LIN {X 0,Y 114.864,Z 300.989,A -85,B 0,C 180,E1 -25798.93,E2 -25798.93} C_VEL
LIN {X 0,Y 114.941,Z 300.979,A -85,B 0,C 180,E1 -25806.506,E2 -25806.506} C_VEL
LIN {X 0,Y 115.012,Z 300.965,A -85,B 0,C 180,E1 -25812.209,E2 -25812.209} C_VEL
LIN {X 0,Y 115.278,Z 300.938,A -85,B 0,C 180,E1 -25817.262,E2 -25817.262} C_VEL
LIN {X 0,Y 115.38,Z 300.924,A -85,B 0,C 180,E1 -25823.002,E2 -25823.002} C_VEL
LIN {X 0,Y 115.988,Z 300.845,A -85,B 0,C 180,E1 -25829.999,E2 -25829.999} C_VEL
LIN {X 0,Y 115.381,Z 300.918,A -85,B 0,C 180,E1 -25836.996,E2 -25836.996} C_VEL
LIN {X 0,Y 115.299,Z 300.934,A -85,B 0,C 180,E1 -25842.784,E2 -25842.784} C_VEL
LIN {X 0,Y 115.207,Z 300.943,A -85,B 0,C 180,E1 -25844.122,E2 -25844.122} C_VEL
LIN {X 0,Y 118.06,Z 309.026,A -85,B 0,C 180,E1 -25845.314,E2 -25845.314} C_VEL
LIN {X 0,Y 124.577,Z 328.009,A -85,B 0,C 180,E1 -25847.836,E2 -25847.836} C_VEL
LIN {X 0,Y 122.385,Z 365.038,A -85,B 0,C 180,E1 -25850.533,E2 -25850.533} C_VEL
LIN {X 0,Y 121.452,Z 375.386,A -85,B 0,C 180,E1 -25851.751,E2 -25851.751} C_VEL
LIN {X 0,Y 120.031,Z 387.44,A -85,B 0,C 180,E1 -25853.894,E2 -25853.894} C_VEL
LIN {X 0,Y 118.866,Z 395.437,A -85,B 0,C 180,E1 -25855.788,E2 -25855.788} C_VEL
LIN {X 0,Y 117.488,Z 403.441,A -85,B 0,C 180,E1 -25858.151,E2 -25858.151} C_VEL
LIN {X 0,Y 116.013,Z 411.202,A -85,B 0,C 180,E1 -25860.991,E2 -25860.991} C_VEL
LIN {X 0,Y 114.685,Z 418.966,A -85,B 0,C 180,E1 -25864.529,E2 -25864.529} C_VEL
LIN {X 0,Y 113.39,Z 426.948,A -85,B 0,C 180,E1 -25869.104,E2 -25869.104} C_VEL
LIN {X 0,Y 112.584,Z 432.701,A -85,B 0,C 180,E1 -25873.365,E2 -25873.365} C_VEL
LIN {X 0,Y 112.223,Z 438.256,A -85,B 0,C 180,E1 -25878.718,E2 -25878.718} C_VEL
LIN {X 0,Y 112.358,Z 440.502,A -85,B 0,C 180,E1 -25881.285,E2 -25881.285} C_VEL
LIN {X 0,Y 113.089,Z 443.74,A -85,B 0,C 180,E1 -25885.996,E2 -25885.996} C_VEL
LIN {X 0,Y 114.462,Z 446.022,A -85,B 0,C 180,E1 -25890.584,E2 -25890.584} C_VEL
LIN {X 0,Y 116.506,Z 447.444,A -85,B 0,C 180,E1 -25895.026,E2 -25895.026} C_VEL
LIN {X 0,Y 119.684,Z 448.034,A -85,B 0,C 180,E1 -25899.97,E2 -25899.97} C_VEL
LIN {X 0,Y 123.835,Z 447.495,A -85,B 0,C 180,E1 -25904.745,E2 -25904.745} C_VEL
LIN {X 0,Y 126.367,Z 446.823,A -85,B 0,C 180,E1 -25907.149,E2 -25907.149} C_VEL
LIN {X 0,Y 130.687,Z 445.002,A -85,B 0,C 180,E1 -25910.719,E2 -25910.719} C_VEL
LIN {X 0,Y 135.629,Z 442.26,A -85,B 0,C 180,E1 -25914.054,E2 -25914.054} C_VEL
LIN {X 0,Y 142.473,Z 437.356,A -85,B 0,C 180,E1 -25917.882,E2 -25917.882} C_VEL
LIN {X 0,Y 147.586,Z 432.947,A -85,B 0,C 180,E1 -25920.364,E2 -25920.364} C_VEL
LIN {X 0,Y 152.954,Z 427.55,A -85,B 0,C 180,E1 -25922.636,E2 -25922.636} C_VEL
LIN {X 0,Y 158.242,Z 421.307,A -85,B 0,C 180,E1 -25924.653,E2 -25924.653} C_VEL
LIN {X 0,Y 163.394,Z 414.148,A -85,B 0,C 180,E1 -25926.442,E2 -25926.442} C_VEL
LIN {X 0,Y 168.811,Z 405.171,A -85,B 0,C 180,E1 -25928.163,E2 -25928.163} C_VEL
LIN {X 0,Y 173.777,Z 394.79,A -85,B 0,C 180,E1 -25929.604,E2 -25929.604} C_VEL
LIN {X 0,Y 177.051,Z 385.976,A -85,B 0,C 180,E1 -25930.574,E2 -25930.574} C_VEL
LIN {X 0,Y 179.653,Z 377.072,A -85,B 0,C 180,E1 -25931.282,E2 -25931.282} C_VEL
LIN {X 0,Y 180.084,Z 375.072,A -85,B 0,C 180,E1 -25931.489,E2 -25931.489} C_VEL
LIN {X 0,Y 178.388,Z 370.508,A -85,B 0,C 180,E1 -25935.201,E2 -25935.201} C_VEL
LIN {X 0,Y 177.063,Z 367.237,A -85,B 0,C 180,E1 -25939.365,E2 -25939.365} C_VEL
LIN {X 0,Y 176.416,Z 366.762,A -85,B 0,C 180,E1 -25943.618,E2 -25943.618} C_VEL
LIN {X 0,Y 176.662,Z 367.081,A -85,B 0,C 180,E1 -25946.725,E2 -25946.725} C_VEL
LIN {X 0,Y 177.162,Z 369.122,A -85,B 0,C 180,E1 -25949.713,E2 -25949.713} C_VEL
LIN {X 0,Y 178.163,Z 373.507,A -85,B 0,C 180,E1 -25953.286,E2 -25953.286} C_VEL
LIN {X 0,Y 179.099,Z 377.548,A -85,B 0,C 180,E1 -25955.579,E2 -25955.579} C_VEL
LIN {X 0,Y 179.509,Z 380.366,A -85,B 0,C 180,E1 -25956.937,E2 -25956.937} C_VEL
LIN {X 0,Y 176.688,Z 390.157,A -85,B 0,C 180,E1 -25957.542,E2 -25957.542} C_VEL
LIN {X 0,Y 173.38,Z 398.961,A -85,B 0,C 180,E1 -25958.264,E2 -25958.264} C_VEL
LIN {X 0,Y 169.107,Z 408.204,A -85,B 0,C 180,E1 -25959.284,E2 -25959.284} C_VEL
LIN {X 0,Y 163.498,Z 418.104,A -85,B 0,C 180,E1 -25960.748,E2 -25960.748} C_VEL
LIN {X 0,Y 157.345,Z 426.798,A -85,B 0,C 180,E1 -25962.526,E2 -25962.526} C_VEL
LIN {X 0,Y 152.186,Z 433.149,A -85,B 0,C 180,E1 -25964.294,E2 -25964.294} C_VEL
LIN {X 0,Y 147.242,Z 438.497,A -85,B 0,C 180,E1 -25966.205,E2 -25966.205} C_VEL
LIN {X 0,Y 142.546,Z 443.022,A -85,B 0,C 180,E1 -25968.274,E2 -25968.274} C_VEL
LIN {X 0,Y 135.864,Z 448.445,A -85,B 0,C 180,E1 -25971.632,E2 -25971.632} C_VEL
LIN {X 0,Y 129.891,Z 452.562,A -85,B 0,C 180,E1 -25975.382,E2 -25975.382} C_VEL
LIN {X 0,Y 124.641,Z 455.495,A -85,B 0,C 180,E1 -25979.506,E2 -25979.506} C_VEL
LIN {X 0,Y 121.618,Z 456.789,A -85,B 0,C 180,E1 -25982.466,E2 -25982.466} C_VEL
LIN {X 0,Y 118.968,Z 457.67,A -85,B 0,C 180,E1 -25985.575,E2 -25985.575} C_VEL
LIN {X 0,Y 116.788,Z 458.13,A -85,B 0,C 180,E1 -25988.836,E2 -25988.836} C_VEL
LIN {X 0,Y 115.116,Z 458.028,A -85,B 0,C 180,E1 -25992.228,E2 -25992.228} C_VEL
LIN {X 0,Y 113.962,Z 457.507,A -85,B 0,C 180,E1 -25995.72,E2 -25995.72} C_VEL
LIN {X 0,Y 113.173,Z 456.575,A -85,B 0,C 180,E1 -25999.264,E2 -25999.264} C_VEL
LIN {X 0,Y 112.949,Z 454.232,A -85,B 0,C 180,E1 -26004.627,E2 -26004.627} C_VEL
LIN {X 0,Y 113.104,Z 452.031,A -85,B 0,C 180,E1 -26008.221,E2 -26008.221} C_VEL
LIN {X 0,Y 113.156,Z 449.13,A -85,B 0,C 180,E1 -26011.78,E2 -26011.78} C_VEL
LIN {X 0,Y 113.228,Z 443.223,A -85,B 0,C 180,E1 -26017.132,E2 -26017.132} C_VEL
LIN {X 0,Y 113.61,Z 438.268,A -85,B 0,C 180,E1 -26020.696,E2 -26020.696} C_VEL
LIN {X 0,Y 114.308,Z 432.256,A -85,B 0,C 180,E1 -26024.238,E2 -26024.238} C_VEL
LIN {X 0,Y 115.483,Z 424.969,A -85,B 0,C 180,E1 -26027.716,E2 -26027.716} C_VEL
LIN {X 0,Y 116.861,Z 417.213,A -85,B 0,C 180,E1 -26030.691,E2 -26030.691} C_VEL
LIN {X 0,Y 118.458,Z 407.592,A -85,B 0,C 180,E1 -26033.608,E2 -26033.608} C_VEL
LIN {X 0,Y 120.245,Z 396.823,A -85,B 0,C 180,E1 -26035.999,E2 -26035.999} C_VEL
LIN {X 0,Y 121.486,Z 386.329,A -85,B 0,C 180,E1 -26037.67,E2 -26037.67} C_VEL
LIN {X 0,Y 122.307,Z 377.143,A -85,B 0,C 180,E1 -26038.69,E2 -26038.69} C_VEL
LIN {X 0,Y 123.167,Z 358.274,A -85,B 0,C 180,E1 -26040.134,E2 -26040.134} C_VEL
LIN {X 0,Y 121.253,Z 329.779,A -85,B 0,C 180,E1 -26042.624,E2 -26042.624} C_VEL
LIN {X 0,Y 120.313,Z 326.084,A -85,B 0,C 180,E1 -26043.058,E2 -26043.058} C_VEL
LIN {X 0,Y 116.845,Z 320.753,A -85,B 0,C 180,E1 -26044.039,E2 -26044.039} C_VEL
LIN {X 0,Y 112.972,Z 315.538,A -85,B 0,C 180,E1 -26045.144,E2 -26045.144} C_VEL
LIN {X 0,Y 111.425,Z 311.965,A -85,B 0,C 180,E1 -26045.734,E2 -26045.734} C_VEL
LIN {X 0,Y 109.288,Z 305.743,A -85,B 0,C 180,E1 -26046.684,E2 -26046.684} C_VEL
LIN {X 0,Y 107.873,Z 301.859,A -85,B 0,C 180,E1 -26047.374,E2 -26047.374} C_VEL
LIN {X 0,Y 107.683,Z 301.879,A -85,B 0,C 180,E1 -26054.113,E2 -26054.113} C_VEL
LIN {X 0,Y 107.687,Z 301.877,A -85,B 0,C 180,E1 -26061.551,E2 -26061.551} C_VEL
LIN {X 0,Y 107.795,Z 301.866,A -85,B 0,C 180,E1 -26068.558,E2 -26068.558} C_VEL
LIN {X 0,Y 107.914,Z 301.852,A -85,B 0,C 180,E1 -26076.995,E2 -26076.995} C_VEL
LIN {X 0,Y 108.031,Z 301.839,A -85,B 0,C 180,E1 -26084.914,E2 -26084.914} C_VEL
LIN {X 0,Y 108.256,Z 301.809,A -85,B 0,C 180,E1 -26088.766,E2 -26088.766} C_VEL
LIN {X 0,Y 108.445,Z 301.784,A -85,B 0,C 180,E1 -26096.281,E2 -26096.281} C_VEL
LIN {X 0,Y 108.942,Z 301.727,A -85,B 0,C 180,E1 -26099.997,E2 -26099.997} C_VEL
LIN {X 0,Y 108.327,Z 301.804,A -85,B 0,C 180,E1 -26107.452,E2 -26107.452} C_VEL
LIN {X 0,Y 108.198,Z 301.813,A -85,B 0,C 180,E1 -26113.012,E2 -26113.012} C_VEL
LIN {X 0,Y 107.909,Z 301.854,A -85,B 0,C 180,E1 -26119.001,E2 -26119.001} C_VEL
LIN {X 0,Y 107.858,Z 301.862,A -85,B 0,C 180,E1 -26124.184,E2 -26124.184} C_VEL
LIN {X 0,Y 107.792,Z 301.87,A -85,B 0,C 180,E1 -26132.049,E2 -26132.049} C_VEL
LIN {X 0,Y 107.73,Z 301.872,A -85,B 0,C 180,E1 -26138.478,E2 -26138.478} C_VEL
LIN {X 0,Y 107.763,Z 301.867,A -85,B 0,C 180,E1 -26145.834,E2 -26145.834} C_VEL
LIN {X 0,Y 107.751,Z 301.876,A -85,B 0,C 180,E1 -26151.502,E2 -26151.502} C_VEL
LIN {X 0,Y 107.806,Z 301.868,A -85,B 0,C 180,E1 -26158.565,E2 -26158.565} C_VEL
LIN {X 0,Y 107.905,Z 301.856,A -85,B 0,C 180,E1 -26166.996,E2 -26166.996} C_VEL
LIN {X 0,Y 108.034,Z 301.839,A -85,B 0,C 180,E1 -26174.917,E2 -26174.917} C_VEL
LIN {X 0,Y 108.281,Z 301.805,A -85,B 0,C 180,E1 -26178.771,E2 -26178.771} C_VEL
LIN {X 0,Y 108.449,Z 301.786,A -85,B 0,C 180,E1 -26186.284,E2 -26186.284} C_VEL
LIN {X 0,Y 108.938,Z 301.723,A -85,B 0,C 180,E1 -26189.999,E2 -26189.999} C_VEL
LIN {X 0,Y 108.321,Z 301.797,A -85,B 0,C 180,E1 -26197.455,E2 -26197.455} C_VEL
LIN {X 0,Y 108.241,Z 301.813,A -85,B 0,C 180,E1 -26202.869,E2 -26202.869} C_VEL
LIN {X 0,Y 117.726,Z 329.232,A -85,B 0,C 180,E1 -26206.93,E2 -26206.93} C_VEL
LIN {X 0,Y 115.492,Z 365.51,A -85,B 0,C 180,E1 -26209.722,E2 -26209.722} C_VEL
LIN {X 0,Y 114.416,Z 376.749,A -85,B 0,C 180,E1 -26211.134,E2 -26211.134} C_VEL
LIN {X 0,Y 112.932,Z 388.546,A -85,B 0,C 180,E1 -26213.43,E2 -26213.43} C_VEL
LIN {X 0,Y 111.623,Z 397.143,A -85,B 0,C 180,E1 -26215.66,E2 -26215.66} C_VEL
LIN {X 0,Y 109.955,Z 405.853,A -85,B 0,C 180,E1 -26218.519,E2 -26218.519} C_VEL
LIN {X 0,Y 108.235,Z 415.195,A -85,B 0,C 180,E1 -26222.428,E2 -26222.428} C_VEL
LIN {X 0,Y 106.799,Z 423.439,A -85,B 0,C 180,E1 -26226.974,E2 -26226.974} C_VEL
LIN {X 0,Y 105.92,Z 429.134,A -85,B 0,C 180,E1 -26230.881,E2 -26230.881} C_VEL
LIN {X 0,Y 105.293,Z 434.326,A -85,B 0,C 180,E1 -26235.26,E2 -26235.26} C_VEL
LIN {X 0,Y 105.173,Z 438.298,A -85,B 0,C 180,E1 -26239.349,E2 -26239.349} C_VEL
LIN {X 0,Y 105.484,Z 441.372,A -85,B 0,C 180,E1 -26243.161,E2 -26243.161} C_VEL
LIN {X 0,Y 106.698,Z 444.823,A -85,B 0,C 180,E1 -26248.899,E2 -26248.899} C_VEL
LIN {X 0,Y 108.938,Z 447.125,A -85,B 0,C 180,E1 -26254.576,E2 -26254.576} C_VEL
LIN {X 0,Y 112.177,Z 448.298,A -85,B 0,C 180,E1 -26260.006,E2 -26260.006} C_VEL
LIN {X 0,Y 116.378,Z 448.344,A -85,B 0,C 180,E1 -26265.059,E2 -26265.059} C_VEL
LIN {X 0,Y 121.731,Z 447.128,A -85,B 0,C 180,E1 -26270.029,E2 -26270.029} C_VEL
LIN {X 0,Y 127.18,Z 444.882,A -85,B 0,C 180,E1 -26274.073,E2 -26274.073} C_VEL
LIN {X 0,Y 133.619,Z 441.3,A -85,B 0,C 180,E1 -26277.875,E2 -26277.875} C_VEL
LIN {X 0,Y 140.594,Z 436.359,A -85,B 0,C 180,E1 -26281.344,E2 -26281.344} C_VEL
LIN {X 0,Y 148.024,Z 429.843,A -85,B 0,C 180,E1 -26284.425,E2 -26284.425} C_VEL
LIN {X 0,Y 153.618,Z 423.846,A -85,B 0,C 180,E1 -26286.477,E2 -26286.477} C_VEL
LIN {X 0,Y 158.966,Z 417.122,A -85,B 0,C 180,E1 -26288.264,E2 -26288.264} C_VEL
LIN {X 0,Y 164.281,Z 409.203,A -85,B 0,C 180,E1 -26289.855,E2 -26289.855} C_VEL
LIN {X 0,Y 168.722,Z 401.241,A -85,B 0,C 180,E1 -26291.109,E2 -26291.109} C_VEL
LIN {X 0,Y 172.503,Z 393.028,A -85,B 0,C 180,E1 -26292.106,E2 -26292.106} C_VEL
LIN {X 0,Y 175.803,Z 383.937,A -85,B 0,C 180,E1 -26293.013,E2 -26293.013} C_VEL
LIN {X 0,Y 177.064,Z 379.788,A -85,B 0,C 180,E1 -26293.348,E2 -26293.348} C_VEL
LIN {X 0,Y 176.232,Z 376.932,A -85,B 0,C 180,E1 -26295.994,E2 -26295.994} C_VEL
LIN {X 0,Y 175.527,Z 374.154,A -85,B 0,C 180,E1 -26299.542,E2 -26299.542} C_VEL
LIN {X 0,Y 174.953,Z 373.704,A -85,B 0,C 180,E1 -26303.687,E2 -26303.687} C_VEL
LIN {X 0,Y 175.186,Z 374.126,A -85,B 0,C 180,E1 -26306.708,E2 -26306.708} C_VEL
LIN {X 0,Y 175.475,Z 375.771,A -85,B 0,C 180,E1 -26309.084,E2 -26309.084} C_VEL
LIN {X 0,Y 176.027,Z 379.665,A -85,B 0,C 180,E1 -26312.378,E2 -26312.378} C_VEL
LIN {X 0,Y 176.544,Z 383.979,A -85,B 0,C 180,E1 -26314.894,E2 -26314.894} C_VEL
LIN {X 0,Y 172.323,Z 396.26,A -85,B 0,C 180,E1 -26315.78,E2 -26315.78} C_VEL
LIN {X 0,Y 168.078,Z 405.486,A -85,B 0,C 180,E1 -26316.663,E2 -26316.663} C_VEL
LIN {X 0,Y 163.359,Z 413.939,A -85,B 0,C 180,E1 -26317.768,E2 -26317.768} C_VEL
LIN {X 0,Y 158.303,Z 421.5,A -85,B 0,C 180,E1 -26319.023,E2 -26319.023} C_VEL
LIN {X 0,Y 151.37,Z 430.324,A -85,B 0,C 180,E1 -26321.023,E2 -26321.023} C_VEL
LIN {X 0,Y 144.794,Z 437.322,A -85,B 0,C 180,E1 -26323.278,E2 -26323.278} C_VEL
LIN {X 0,Y 139.815,Z 441.962,A -85,B 0,C 180,E1 -26325.275,E2 -26325.275} C_VEL
LIN {X 0,Y 132.692,Z 447.497,A -85,B 0,C 180,E1 -26328.545,E2 -26328.545} C_VEL
LIN {X 0,Y 126.141,Z 451.703,A -85,B 0,C 180,E1 -26332.204,E2 -26332.204} C_VEL
LIN {X 0,Y 122.164,Z 453.868,A -85,B 0,C 180,E1 -26334.882,E2 -26334.882} C_VEL
LIN {X 0,Y 118.571,Z 455.571,A -85,B 0,C 180,E1 -26337.763,E2 -26337.763} C_VEL
LIN {X 0,Y 115.374,Z 456.695,A -85,B 0,C 180,E1 -26340.837,E2 -26340.837} C_VEL
LIN {X 0,Y 112.549,Z 457.369,A -85,B 0,C 180,E1 -26344.082,E2 -26344.082} C_VEL
LIN {X 0,Y 110.187,Z 457.652,A -85,B 0,C 180,E1 -26347.501,E2 -26347.501} C_VEL
LIN {X 0,Y 108.371,Z 457.513,A -85,B 0,C 180,E1 -26351.081,E2 -26351.081} C_VEL
LIN {X 0,Y 107.114,Z 456.823,A -85,B 0,C 180,E1 -26354.786,E2 -26354.786} C_VEL
LIN {X 0,Y 106.233,Z 455.696,A -85,B 0,C 180,E1 -26358.554,E2 -26358.554} C_VEL
LIN {X 0,Y 105.948,Z 453.139,A -85,B 0,C 180,E1 -26364.305,E2 -26364.305} C_VEL
LIN {X 0,Y 106.133,Z 450.763,A -85,B 0,C 180,E1 -26368.104,E2 -26368.104} C_VEL
LIN {X 0,Y 106.149,Z 447.7,A -85,B 0,C 180,E1 -26371.898,E2 -26371.898} C_VEL
LIN {X 0,Y 106.18,Z 443.174,A -85,B 0,C 180,E1 -26376.266,E2 -26376.266} C_VEL
LIN {X 0,Y 106.545,Z 437.759,A -85,B 0,C 180,E1 -26380.452,E2 -26380.452} C_VEL
LIN {X 0,Y 107.237,Z 431.73,A -85,B 0,C 180,E1 -26384.228,E2 -26384.228} C_VEL
LIN {X 0,Y 108.422,Z 424.419,A -85,B 0,C 180,E1 -26387.933,E2 -26387.933} C_VEL
LIN {X 0,Y 109.848,Z 416.641,A -85,B 0,C 180,E1 -26391.093,E2 -26391.093} C_VEL
LIN {X 0,Y 111.489,Z 406.981,A -85,B 0,C 180,E1 -26394.189,E2 -26394.189} C_VEL
LIN {X 0,Y 113.326,Z 396.093,A -85,B 0,C 180,E1 -26396.719,E2 -26396.719} C_VEL
LIN {X 0,Y 114.559,Z 386.165,A -85,B 0,C 180,E1 -26398.389,E2 -26398.389} C_VEL
LIN {X 0,Y 115.451,Z 376.307,A -85,B 0,C 180,E1 -26399.542,E2 -26399.542} C_VEL
LIN {X 0,Y 116.301,Z 358.488,A -85,B 0,C 180,E1 -26400.978,E2 -26400.978} C_VEL
LIN {X 0,Y 113.92,Z 320.888,A -85,B 0,C 180,E1 -26404.509,E2 -26404.509} C_VEL
LIN {X 0,Y 111.425,Z 311.965,A -85,B 0,C 180,E1 -26405.734,E2 -26405.734} C_VEL
LIN {X 0,Y 110.153,Z 308.851,A -85,B 0,C 180,E1 -26406.532,E2 -26406.532} C_VEL
LIN {X 0,Y 108.481,Z 306.509,A -85,B 0,C 180,E1 -26407.797,E2 -26407.797} C_VEL
LIN {X 0,Y 106.664,Z 304.831,A -85,B 0,C 180,E1 -26409.398,E2 -26409.398} C_VEL
LIN {X 0,Y 104.071,Z 303.42,A -85,B 0,C 180,E1 -26412.26,E2 -26412.26} C_VEL
LIN {X 0,Y 101.917,Z 302.856,A -85,B 0,C 180,E1 -26415.615,E2 -26415.615} C_VEL
LIN {X 0,Y 100.633,Z 302.756,A -85,B 0,C 180,E1 -26420.407,E2 -26420.407} C_VEL
LIN {X 0,Y 100.691,Z 302.754,A -85,B 0,C 180,E1 -26426.884,E2 -26426.884} C_VEL
LIN {X 0,Y 100.789,Z 302.743,A -85,B 0,C 180,E1 -26435.264,E2 -26435.264} C_VEL
LIN {X 0,Y 100.818,Z 302.733,A -85,B 0,C 180,E1 -26439.598,E2 -26439.598} C_VEL
LIN {X 0,Y 101.105,Z 302.696,A -85,B 0,C 180,E1 -26446.696,E2 -26446.696} C_VEL
LIN {X 0,Y 101.243,Z 302.686,A -85,B 0,C 180,E1 -26452.016,E2 -26452.016} C_VEL
LIN {X 0,Y 101.865,Z 302.609,A -85,B 0,C 180,E1 -26459.997,E2 -26459.997} C_VEL
LIN {X 0,Y 101.266,Z 302.684,A -85,B 0,C 180,E1 -26467.975,E2 -26467.975} C_VEL
LIN {X 0,Y 101.123,Z 302.695,A -85,B 0,C 180,E1 -26473.347,E2 -26473.347} C_VEL
LIN {X 0,Y 100.819,Z 302.731,A -85,B 0,C 180,E1 -26480.395,E2 -26480.395} C_VEL
LIN {X 0,Y 100.772,Z 302.745,A -85,B 0,C 180,E1 -26484.955,E2 -26484.955} C_VEL
LIN {X 0,Y 100.699,Z 302.754,A -85,B 0,C 180,E1 -26493.122,E2 -26493.122} C_VEL
LIN {X 0,Y 100.683,Z 302.753,A -85,B 0,C 180,E1 -26499.84,E2 -26499.84} C_VEL
LIN {X 0,Y 100.729,Z 302.743,A -85,B 0,C 180,E1 -26505.756,E2 -26505.756} C_VEL
LIN {X 0,Y 100.691,Z 302.755,A -85,B 0,C 180,E1 -26511.084,E2 -26511.084} C_VEL
LIN {X 0,Y 100.703,Z 302.751,A -85,B 0,C 180,E1 -26516.867,E2 -26516.867} C_VEL
LIN {X 0,Y 100.781,Z 302.741,A -85,B 0,C 180,E1 -26525.265,E2 -26525.265} C_VEL
LIN {X 0,Y 100.812,Z 302.737,A -85,B 0,C 180,E1 -26529.6,E2 -26529.6} C_VEL
LIN {X 0,Y 101.181,Z 302.691,A -85,B 0,C 180,E1 -26537.972,E2 -26537.972} C_VEL
LIN {X 0,Y 101.259,Z 302.681,A -85,B 0,C 180,E1 -26542.02,E2 -26542.02} C_VEL
LIN {X 0,Y 101.862,Z 302.604,A -85,B 0,C 180,E1 -26549.999,E2 -26549.999} C_VEL
LIN {X 0,Y 101.209,Z 302.69,A -85,B 0,C 180,E1 -26559.996,E2 -26559.996} C_VEL
LIN {X 0,Y 101.23,Z 302.695,A -85,B 0,C 180,E1 -26561.512,E2 -26561.512} C_VEL
LIN {X 0,Y 109.715,Z 327.024,A -85,B 0,C 180,E1 -26565.45,E2 -26565.45} C_VEL
LIN {X 0,Y 110.926,Z 330.649,A -85,B 0,C 180,E1 -26565.97,E2 -26565.97} C_VEL
LIN {X 0,Y 108.569,Z 366.195,A -85,B 0,C 180,E1 -26568.883,E2 -26568.883} C_VEL
LIN {X 0,Y 107.508,Z 376.881,A -85,B 0,C 180,E1 -26570.32,E2 -26570.32} C_VEL
LIN {X 0,Y 105.93,Z 388.713,A -85,B 0,C 180,E1 -26572.748,E2 -26572.748} C_VEL
LIN {X 0,Y 104.582,Z 397.271,A -85,B 0,C 180,E1 -26575.099,E2 -26575.099} C_VEL
LIN {X 0,Y 102.954,Z 405.585,A -85,B 0,C 180,E1 -26577.973,E2 -26577.973} C_VEL
LIN {X 0,Y 101.47,Z 413.261,A -85,B 0,C 180,E1 -26581.294,E2 -26581.294} C_VEL
LIN {X 0,Y 99.879,Z 422.113,A -85,B 0,C 180,E1 -26586.119,E2 -26586.119} C_VEL
LIN {X 0,Y 98.836,Z 428.765,A -85,B 0,C 180,E1 -26590.815,E2 -26590.815} C_VEL
LIN {X 0,Y 98.205,Z 434.277,A -85,B 0,C 180,E1 -26595.694,E2 -26595.694} C_VEL
LIN {X 0,Y 98.105,Z 438.154,A -85,B 0,C 180,E1 -26599.859,E2 -26599.859} C_VEL
LIN {X 0,Y 98.717,Z 442.149,A -85,B 0,C 180,E1 -26605.286,E2 -26605.286} C_VEL
LIN {X 0,Y 100.004,Z 445.115,A -85,B 0,C 180,E1 -26610.536,E2 -26610.536} C_VEL
LIN {X 0,Y 102.121,Z 447.209,A -85,B 0,C 180,E1 -26615.615,E2 -26615.615} C_VEL
LIN {X 0,Y 104.949,Z 448.471,A -85,B 0,C 180,E1 -26620.442,E2 -26620.442} C_VEL
LIN {X 0,Y 108.915,Z 448.907,A -85,B 0,C 180,E1 -26625.437,E2 -26625.437} C_VEL
LIN {X 0,Y 114.032,Z 448.286,A -85,B 0,C 180,E1 -26630.426,E2 -26630.426} C_VEL
LIN {X 0,Y 119.94,Z 446.542,A -85,B 0,C 180,E1 -26634.933,E2 -26634.933} C_VEL
LIN {X 0,Y 126.523,Z 443.647,A -85,B 0,C 180,E1 -26638.897,E2 -26638.897} C_VEL
LIN {X 0,Y 134.811,Z 438.573,A -85,B 0,C 180,E1 -26642.991,E2 -26642.991} C_VEL
LIN {X 0,Y 141.433,Z 433.5,A -85,B 0,C 180,E1 -26645.706,E2 -26645.706} C_VEL
LIN {X 0,Y 146.639,Z 428.808,A -85,B 0,C 180,E1 -26647.576,E2 -26647.576} C_VEL
LIN {X 0,Y 152.262,Z 422.841,A -85,B 0,C 180,E1 -26649.454,E2 -26649.454} C_VEL
LIN {X 0,Y 157.501,Z 416.358,A -85,B 0,C 180,E1 -26650.993,E2 -26650.993} C_VEL
LIN {X 0,Y 162.848,Z 408.475,A -85,B 0,C 180,E1 -26652.464,E2 -26652.464} C_VEL
LIN {X 0,Y 168.135,Z 399.051,A -85,B 0,C 180,E1 -26653.798,E2 -26653.798} C_VEL
LIN {X 0,Y 172.792,Z 388.253,A -85,B 0,C 180,E1 -26654.939,E2 -26654.939} C_VEL
LIN {X 0,Y 174.007,Z 384.648,A -85,B 0,C 180,E1 -26655.317,E2 -26655.317} C_VEL
LIN {X 0,Y 173.887,Z 383.473,A -85,B 0,C 180,E1 -26656.436,E2 -26656.436} C_VEL
LIN {X 0,Y 173.457,Z 380.938,A -85,B 0,C 180,E1 -26659.785,E2 -26659.785} C_VEL
LIN {X 0,Y 173.031,Z 380.56,A -85,B 0,C 180,E1 -26663.966,E2 -26663.966} C_VEL
LIN {X 0,Y 173.236,Z 380.955,A -85,B 0,C 180,E1 -26666.506,E2 -26666.506} C_VEL
LIN {X 0,Y 173.333,Z 382.439,A -85,B 0,C 180,E1 -26668.643,E2 -26668.643} C_VEL
LIN {X 0,Y 173.564,Z 384.731,A -85,B 0,C 180,E1 -26670.725,E2 -26670.725} C_VEL
LIN {X 0,Y 173.614,Z 387.116,A -85,B 0,C 180,E1 -26672.408,E2 -26672.408} C_VEL
LIN {X 0,Y 173.404,Z 388.506,A -85,B 0,C 180,E1 -26672.952,E2 -26672.952} C_VEL
LIN {X 0,Y 169.754,Z 397.736,A -85,B 0,C 180,E1 -26673.602,E2 -26673.602} C_VEL
LIN {X 0,Y 165.16,Z 407.074,A -85,B 0,C 180,E1 -26674.491,E2 -26674.491} C_VEL
LIN {X 0,Y 159.199,Z 416.929,A -85,B 0,C 180,E1 -26675.791,E2 -26675.791} C_VEL
LIN {X 0,Y 152.562,Z 425.648,A -85,B 0,C 180,E1 -26677.381,E2 -26677.381} C_VEL
LIN {X 0,Y 146.884,Z 432.024,A -85,B 0,C 180,E1 -26678.969,E2 -26678.969} C_VEL
LIN {X 0,Y 140.086,Z 438.549,A -85,B 0,C 180,E1 -26681.192,E2 -26681.192} C_VEL
LIN {X 0,Y 134.896,Z 442.877,A -85,B 0,C 180,E1 -26683.167,E2 -26683.167} C_VEL
LIN {X 0,Y 127.479,Z 448.131,A -85,B 0,C 180,E1 -26686.441,E2 -26686.441} C_VEL
LIN {X 0,Y 122.867,Z 450.889,A -85,B 0,C 180,E1 -26688.87,E2 -26688.87} C_VEL
LIN {X 0,Y 116.433,Z 454.016,A -85,B 0,C 180,E1 -26692.873,E2 -26692.873} C_VEL
LIN {X 0,Y 112.622,Z 455.504,A -85,B 0,C 180,E1 -26695.833,E2 -26695.833} C_VEL
LIN {X 0,Y 109.235,Z 456.566,A -85,B 0,C 180,E1 -26699.024,E2 -26699.024} C_VEL
LIN {X 0,Y 106.218,Z 457.073,A -85,B 0,C 180,E1 -26702.41,E2 -26702.41} C_VEL
LIN {X 0,Y 103.658,Z 457.146,A -85,B 0,C 180,E1 -26705.998,E2 -26705.998} C_VEL
LIN {X 0,Y 101.681,Z 456.84,A -85,B 0,C 180,E1 -26709.784,E2 -26709.784} C_VEL
LIN {X 0,Y 100.288,Z 456.107,A -85,B 0,C 180,E1 -26713.722,E2 -26713.722} C_VEL
LIN {X 0,Y 99.313,Z 454.806,A -85,B 0,C 180,E1 -26717.744,E2 -26717.744} C_VEL
LIN {X 0,Y 98.957,Z 452.068,A -85,B 0,C 180,E1 -26723.899,E2 -26723.899} C_VEL
LIN {X 0,Y 99.154,Z 449.484,A -85,B 0,C 180,E1 -26727.97,E2 -26727.97} C_VEL
LIN {X 0,Y 99.161,Z 446.19,A -85,B 0,C 180,E1 -26732.032,E2 -26732.032} C_VEL
LIN {X 0,Y 99.172,Z 441.414,A -85,B 0,C 180,E1 -26736.698,E2 -26736.698} C_VEL
LIN {X 0,Y 99.641,Z 435.711,A -85,B 0,C 180,E1 -26741.185,E2 -26741.185} C_VEL
LIN {X 0,Y 100.704,Z 427.689,A -85,B 0,C 180,E1 -26746.21,E2 -26746.21} C_VEL
LIN {X 0,Y 102.412,Z 418.375,A -85,B 0,C 180,E1 -26750.592,E2 -26750.592} C_VEL
LIN {X 0,Y 103.792,Z 410.675,A -85,B 0,C 180,E1 -26753.442,E2 -26753.442} C_VEL
LIN {X 0,Y 105.129,Z 402.866,A -85,B 0,C 180,E1 -26755.756,E2 -26755.756} C_VEL
LIN {X 0,Y 106.597,Z 394.192,A -85,B 0,C 180,E1 -26757.752,E2 -26757.752} C_VEL
LIN {X 0,Y 107.779,Z 384.556,A -85,B 0,C 180,E1 -26759.413,E2 -26759.413} C_VEL
LIN {X 0,Y 108.674,Z 374.382,A -85,B 0,C 180,E1 -26760.616,E2 -26760.616} C_VEL
LIN {X 0,Y 109.46,Z 358.779,A -85,B 0,C 180,E1 -26761.925,E2 -26761.925} C_VEL
LIN {X 0,Y 107.133,Z 322.026,A -85,B 0,C 180,E1 -26765.6,E2 -26765.6} C_VEL
LIN {X 0,Y 103.495,Z 309.671,A -85,B 0,C 180,E1 -26767.456,E2 -26767.456} C_VEL
LIN {X 0,Y 100.801,Z 303.194,A -85,B 0,C 180,E1 -26768.666,E2 -26768.666} C_VEL
LIN {X 0,Y 100.723,Z 302.751,A -85,B 0,C 180,E1 -26768.902,E2 -26768.902} C_VEL
LIN {X 0,Y 100.65,Z 302.759,A -85,B 0,C 180,E1 -26775.708,E2 -26775.708} C_VEL
LIN {X 0,Y 100.633,Z 302.756,A -85,B 0,C 180,E1 -26780.407,E2 -26780.407} C_VEL
LIN {X 0,Y 99.942,Z 302.846,A -85,B 0,C 180,E1 -26783.749,E2 -26783.749} C_VEL
LIN {X 0,Y 98.409,Z 303.039,A -85,B 0,C 180,E1 -26787.062,E2 -26787.062} C_VEL
LIN {X 0,Y 94.006,Z 303.585,A -85,B 0,C 180,E1 -26796.318,E2 -26796.318} C_VEL
LIN {X 0,Y 93.668,Z 303.618,A -85,B 0,C 180,E1 -26798.78,E2 -26798.78} C_VEL
LIN {X 0,Y 94.069,Z 303.572,A -85,B 0,C 180,E1 -26807.045,E2 -26807.045} C_VEL
LIN {X 0,Y 94.177,Z 303.567,A -85,B 0,C 180,E1 -26811.413,E2 -26811.413} C_VEL
LIN {X 0,Y 94.791,Z 303.49,A -85,B 0,C 180,E1 -26819.996,E2 -26819.996} C_VEL
LIN {X 0,Y 94.199,Z 303.563,A -85,B 0,C 180,E1 -26828.578,E2 -26828.578} C_VEL
LIN {X 0,Y 94.041,Z 303.578,A -85,B 0,C 180,E1 -26833.704,E2 -26833.704} C_VEL
LIN {X 0,Y 93.694,Z 303.621,A -85,B 0,C 180,E1 -26842.023,E2 -26842.023} C_VEL
LIN {X 0,Y 93.621,Z 303.634,A -85,B 0,C 180,E1 -26846.766,E2 -26846.766} C_VEL
LIN {X 0,Y 93.601,Z 303.637,A -85,B 0,C 180,E1 -26854.317,E2 -26854.317} C_VEL
LIN {X 0,Y 93.608,Z 303.637,A -85,B 0,C 180,E1 -26862.504,E2 -26862.504} C_VEL
LIN {X 0,Y 93.624,Z 303.633,A -85,B 0,C 180,E1 -26868.642,E2 -26868.642} C_VEL
LIN {X 0,Y 93.609,Z 303.63,A -85,B 0,C 180,E1 -26875.669,E2 -26875.669} C_VEL
LIN {X 0,Y 93.664,Z 303.624,A -85,B 0,C 180,E1 -26884.202,E2 -26884.202} C_VEL
LIN {X 0,Y 93.689,Z 303.627,A -85,B 0,C 180,E1 -26887.971,E2 -26887.971} C_VEL
LIN {X 0,Y 94.085,Z 303.577,A -85,B 0,C 180,E1 -26897.05,E2 -26897.05} C_VEL
LIN {X 0,Y 94.192,Z 303.559,A -85,B 0,C 180,E1 -26901.417,E2 -26901.417} C_VEL
LIN {X 0,Y 94.788,Z 303.485,A -85,B 0,C 180,E1 -26909.999,E2 -26909.999} C_VEL
LIN {X 0,Y 94.184,Z 303.621,A -85,B 0,C 180,E1 -26919.935,E2 -26919.935} C_VEL
LIN {X 0,Y 101.629,Z 324.517,A -85,B 0,C 180,E1 -26923.736,E2 -26923.736} C_VEL
LIN {X 0,Y 104.051,Z 332.19,A -85,B 0,C 180,E1 -26924.933,E2 -26924.933} C_VEL
LIN {X 0,Y 101.715,Z 366.427,A -85,B 0,C 180,E1 -26927.917,E2 -26927.917} C_VEL
LIN {X 0,Y 100.374,Z 378.614,A -85,B 0,C 180,E1 -26929.69,E2 -26929.69} C_VEL
LIN {X 0,Y 98.959,Z 388.967,A -85,B 0,C 180,E1 -26932.003,E2 -26932.003} C_VEL
LIN {X 0,Y 97.593,Z 397.115,A -85,B 0,C 180,E1 -26934.361,E2 -26934.361} C_VEL
LIN {X 0,Y 96.11,Z 404.37,A -85,B 0,C 180,E1 -26936.952,E2 -26936.952} C_VEL
LIN {X 0,Y 94.525,Z 412.39,A -85,B 0,C 180,E1 -26940.54,E2 -26940.54} C_VEL
LIN {X 0,Y 93.354,Z 418.852,A -85,B 0,C 180,E1 -26944.101,E2 -26944.101} C_VEL
LIN {X 0,Y 92.153,Z 425.721,A -85,B 0,C 180,E1 -26948.781,E2 -26948.781} C_VEL
LIN {X 0,Y 91.294,Z 431.706,A -85,B 0,C 180,E1 -26953.853,E2 -26953.853} C_VEL
LIN {X 0,Y 91.018,Z 436.118,A -85,B 0,C 180,E1 -26958.442,E2 -26958.442} C_VEL
LIN {X 0,Y 91.504,Z 441.017,A -85,B 0,C 180,E1 -26964.752,E2 -26964.752} C_VEL
LIN {X 0,Y 92.791,Z 444.457,A -85,B 0,C 180,E1 -26970.512,E2 -26970.512} C_VEL
LIN {X 0,Y 93.959,Z 446.004,A -85,B 0,C 180,E1 -26973.837,E2 -26973.837} C_VEL
LIN {X 0,Y 97.177,Z 448.193,A -85,B 0,C 180,E1 -26980.075,E2 -26980.075} C_VEL
LIN {X 0,Y 101.449,Z 449.268,A -85,B 0,C 180,E1 -26985.89,E2 -26985.89} C_VEL
LIN {X 0,Y 106.679,Z 449.233,A -85,B 0,C 180,E1 -26991.174,E2 -26991.174} C_VEL
LIN {X 0,Y 113.516,Z 447.762,A -85,B 0,C 180,E1 -26996.453,E2 -26996.453} C_VEL
LIN {X 0,Y 119.472,Z 445.63,A -85,B 0,C 180,E1 -27000.08,E2 -27000.08} C_VEL
LIN {X 0,Y 126.765,Z 442.066,A -85,B 0,C 180,E1 -27003.708,E2 -27003.708} C_VEL
LIN {X 0,Y 132.322,Z 438.67,A -85,B 0,C 180,E1 -27006.1,E2 -27006.1} C_VEL
LIN {X 0,Y 139.388,Z 433.448,A -85,B 0,C 180,E1 -27008.702,E2 -27008.702} C_VEL
LIN {X 0,Y 144.627,Z 428.839,A -85,B 0,C 180,E1 -27010.428,E2 -27010.428} C_VEL
LIN {X 0,Y 151.085,Z 422.177,A -85,B 0,C 180,E1 -27012.36,E2 -27012.36} C_VEL
LIN {X 0,Y 158.364,Z 413.174,A -85,B 0,C 180,E1 -27014.237,E2 -27014.237} C_VEL
LIN {X 0,Y 164.392,Z 403.606,A -85,B 0,C 180,E1 -27015.685,E2 -27015.685} C_VEL
LIN {X 0,Y 169.072,Z 394.321,A -85,B 0,C 180,E1 -27016.745,E2 -27016.745} C_VEL
LIN {X 0,Y 170.937,Z 390.096,A -85,B 0,C 180,E1 -27017.141,E2 -27017.141} C_VEL
LIN {X 0,Y 171.041,Z 389.404,A -85,B 0,C 180,E1 -27017.544,E2 -27017.544} C_VEL
LIN {X 0,Y 170.904,Z 388.246,A -85,B 0,C 180,E1 -27019.209,E2 -27019.209} C_VEL
LIN {X 0,Y 170.792,Z 387.317,A -85,B 0,C 180,E1 -27021.739,E2 -27021.739} C_VEL
LIN {X 0,Y 170.79,Z 387.347,A -85,B 0,C 180,E1 -27025.141,E2 -27025.141} C_VEL
LIN {X 0,Y 170.87,Z 387.973,A -85,B 0,C 180,E1 -27026.902,E2 -27026.902} C_VEL
LIN {X 0,Y 170.792,Z 391.193,A -85,B 0,C 180,E1 -27030.218,E2 -27030.218} C_VEL
LIN {X 0,Y 170.778,Z 391.803,A -85,B 0,C 180,E1 -27030.672,E2 -27030.672} C_VEL
LIN {X 0,Y 169.859,Z 394.284,A -85,B 0,C 180,E1 -27030.981,E2 -27030.981} C_VEL
LIN {X 0,Y 165.268,Z 403.838,A -85,B 0,C 180,E1 -27031.737,E2 -27031.737} C_VEL
LIN {X 0,Y 160.607,Z 411.818,A -85,B 0,C 180,E1 -27032.613,E2 -27032.613} C_VEL
LIN {X 0,Y 155.982,Z 418.536,A -85,B 0,C 180,E1 -27033.538,E2 -27033.538} C_VEL
LIN {X 0,Y 149.914,Z 426.001,A -85,B 0,C 180,E1 -27034.878,E2 -27034.878} C_VEL
LIN {X 0,Y 144.035,Z 432.252,A -85,B 0,C 180,E1 -27036.383,E2 -27036.383} C_VEL
LIN {X 0,Y 136.939,Z 438.68,A -85,B 0,C 180,E1 -27038.498,E2 -27038.498} C_VEL
LIN {X 0,Y 130.188,Z 443.867,A -85,B 0,C 180,E1 -27040.91,E2 -27040.91} C_VEL
LIN {X 0,Y 122.453,Z 448.802,A -85,B 0,C 180,E1 -27044.161,E2 -27044.161} C_VEL
LIN {X 0,Y 115.28,Z 452.427,A -85,B 0,C 180,E1 -27047.888,E2 -27047.888} C_VEL
LIN {X 0,Y 110.863,Z 454.174,A -85,B 0,C 180,E1 -27050.661,E2 -27050.661} C_VEL
LIN {X 0,Y 106.816,Z 455.434,A -85,B 0,C 180,E1 -27053.692,E2 -27053.692} C_VEL
LIN {X 0,Y 103.221,Z 456.293,A -85,B 0,C 180,E1 -27056.998,E2 -27056.998} C_VEL
LIN {X 0,Y 99.991,Z 456.745,A -85,B 0,C 180,E1 -27060.53,E2 -27060.53} C_VEL
LIN {X 0,Y 97.211,Z 456.641,A -85,B 0,C 180,E1 -27064.294,E2 -27064.294} C_VEL
LIN {X 0,Y 95.055,Z 456.13,A -85,B 0,C 180,E1 -27068.306,E2 -27068.306} C_VEL
LIN {X 0,Y 93.523,Z 455.24,A -85,B 0,C 180,E1 -27072.508,E2 -27072.508} C_VEL
LIN {X 0,Y 92.423,Z 453.88,A -85,B 0,C 180,E1 -27076.815,E2 -27076.815} C_VEL
LIN {X 0,Y 91.991,Z 450.938,A -85,B 0,C 180,E1 -27083.336,E2 -27083.336} C_VEL
LIN {X 0,Y 92.175,Z 448.193,A -85,B 0,C 180,E1 -27087.816,E2 -27087.816} C_VEL
LIN {X 0,Y 92.124,Z 443.729,A -85,B 0,C 180,E1 -27093.281,E2 -27093.281} C_VEL
LIN {X 0,Y 92.299,Z 437.863,A -85,B 0,C 180,E1 -27098.76,E2 -27098.76} C_VEL
LIN {X 0,Y 92.922,Z 432.082,A -85,B 0,C 180,E1 -27103.115,E2 -27103.115} C_VEL
LIN {X 0,Y 93.975,Z 425.02,A -85,B 0,C 180,E1 -27107.407,E2 -27107.407} C_VEL
LIN {X 0,Y 95.411,Z 417.577,A -85,B 0,C 180,E1 -27111.045,E2 -27111.045} C_VEL
LIN {X 0,Y 96.83,Z 409.788,A -85,B 0,C 180,E1 -27114.097,E2 -27114.097} C_VEL
LIN {X 0,Y 98.249,Z 401.891,A -85,B 0,C 180,E1 -27116.557,E2 -27116.557} C_VEL
LIN {X 0,Y 99.928,Z 391.94,A -85,B 0,C 180,E1 -27118.916,E2 -27118.916} C_VEL
LIN {X 0,Y 101.36,Z 380.093,A -85,B 0,C 180,E1 -27120.9,E2 -27120.9} C_VEL
LIN {X 0,Y 102.592,Z 361.843,A -85,B 0,C 180,E1 -27122.648,E2 -27122.648} C_VEL
LIN {X 0,Y 100.528,Z 323.725,A -85,B 0,C 180,E1 -27126.694,E2 -27126.694} C_VEL
LIN {X 0,Y 97.095,Z 312.114,A -85,B 0,C 180,E1 -27128.611,E2 -27128.611} C_VEL
LIN {X 0,Y 93.641,Z 303.83,A -85,B 0,C 180,E1 -27130.332,E2 -27130.332} C_VEL
LIN {X 0,Y 93.536,Z 303.645,A -85,B 0,C 180,E1 -27138.709,E2 -27138.709} C_VEL
LIN {X 0,Y 93.588,Z 303.641,A -85,B 0,C 180,E1 -27145.695,E2 -27145.695} C_VEL
LIN {X 0,Y 93.671,Z 303.629,A -85,B 0,C 180,E1 -27154.203,E2 -27154.203} C_VEL
LIN {X 0,Y 93.668,Z 303.618,A -85,B 0,C 180,E1 -27158.78,E2 -27158.78} C_VEL
LIN {X 0,Y 92.956,Z 303.718,A -85,B 0,C 180,E1 -27162.376,E2 -27162.376} C_VEL
LIN {X 0,Y 91.41,Z 303.91,A -85,B 0,C 180,E1 -27165.948,E2 -27165.948} C_VEL
LIN {X 0,Y 87.496,Z 304.391,A -85,B 0,C 180,E1 -27175.987,E2 -27175.987} C_VEL
LIN {X 0,Y 87.506,Z 304.388,A -85,B 0,C 180,E1 -27178.629,E2 -27178.629} C_VEL
LIN {X 0,Y 87.717,Z 304.371,A -85,B 0,C 180,E1 -27179.996,E2 -27179.996} C_VEL
LIN {X 0,Y 87.107,Z 304.447,A -85,B 0,C 180,E1 -27189.282,E2 -27189.282} C_VEL
LIN {X 0,Y 86.949,Z 304.462,A -85,B 0,C 180,E1 -27194.083,E2 -27194.083} C_VEL
LIN {X 0,Y 86.586,Z 304.512,A -85,B 0,C 180,E1 -27203.939,E2 -27203.939} C_VEL
LIN {X 0,Y 86.476,Z 304.518,A -85,B 0,C 180,E1 -27209.18,E2 -27209.18} C_VEL
LIN {X 0,Y 86.524,Z 304.516,A -85,B 0,C 180,E1 -27215.683,E2 -27215.683} C_VEL
LIN {X 0,Y 86.54,Z 304.517,A -85,B 0,C 180,E1 -27223.038,E2 -27223.038} C_VEL
LIN {X 0,Y 86.549,Z 304.516,A -85,B 0,C 180,E1 -27229.486,E2 -27229.486} C_VEL
LIN {X 0,Y 86.557,Z 304.507,A -85,B 0,C 180,E1 -27235.363,E2 -27235.363} C_VEL
LIN {X 0,Y 86.581,Z 304.505,A -85,B 0,C 180,E1 -27243.23,E2 -27243.23} C_VEL
LIN {X 0,Y 86.642,Z 304.498,A -85,B 0,C 180,E1 -27251.066,E2 -27251.066} C_VEL
LIN {X 0,Y 86.964,Z 304.465,A -85,B 0,C 180,E1 -27255.968,E2 -27255.968} C_VEL
LIN {X 0,Y 87.101,Z 304.44,A -85,B 0,C 180,E1 -27260.712,E2 -27260.712} C_VEL
LIN {X 0,Y 87.716,Z 304.365,A -85,B 0,C 180,E1 -27269.999,E2 -27269.999} C_VEL
LIN {X 0,Y 87.159,Z 304.434,A -85,B 0,C 180,E1 -27278.111,E2 -27278.111} C_VEL
LIN {X 0,Y 89.669,Z 311.03,A -85,B 0,C 180,E1 -27279.604,E2 -27279.604} C_VEL
LIN {X 0,Y 96.258,Z 330.029,A -85,B 0,C 180,E1 -27283.167,E2 -27283.167} C_VEL
LIN {X 0,Y 97.222,Z 333.154,A -85,B 0,C 180,E1 -27283.693,E2 -27283.693} C_VEL
LIN {X 0,Y 94.874,Z 366.766,A -85,B 0,C 180,E1 -27286.823,E2 -27286.823} C_VEL
LIN {X 0,Y 93.503,Z 378.519,A -85,B 0,C 180,E1 -27288.628,E2 -27288.628} C_VEL
LIN {X 0,Y 91.887,Z 389.671,A -85,B 0,C 180,E1 -27291.302,E2 -27291.302} C_VEL
LIN {X 0,Y 90.306,Z 398.504,A -85,B 0,C 180,E1 -27294.114,E2 -27294.114} C_VEL
LIN {X 0,Y 88.697,Z 405.975,A -85,B 0,C 180,E1 -27297.102,E2 -27297.102} C_VEL
LIN {X 0,Y 86.931,Z 415.024,A -85,B 0,C 180,E1 -27301.7,E2 -27301.7} C_VEL
LIN {X 0,Y 85.326,Z 423.875,A -85,B 0,C 180,E1 -27307.562,E2 -27307.562} C_VEL
LIN {X 0,Y 84.311,Z 430.48,A -85,B 0,C 180,E1 -27313.278,E2 -27313.278} C_VEL
LIN {X 0,Y 83.975,Z 435.689,A -85,B 0,C 180,E1 -27318.868,E2 -27318.868} C_VEL
LIN {X 0,Y 84.621,Z 441.049,A -85,B 0,C 180,E1 -27326.149,E2 -27326.149} C_VEL
LIN {X 0,Y 86.487,Z 445.09,A -85,B 0,C 180,E1 -27333.358,E2 -27333.358} C_VEL
LIN {X 0,Y 89.67,Z 447.841,A -85,B 0,C 180,E1 -27340.131,E2 -27340.131} C_VEL
LIN {X 0,Y 94.594,Z 449.468,A -85,B 0,C 180,E1 -27347.125,E2 -27347.125} C_VEL
LIN {X 0,Y 99.349,Z 449.8,A -85,B 0,C 180,E1 -27352.026,E2 -27352.026} C_VEL
LIN {X 0,Y 105.558,Z 449.134,A -85,B 0,C 180,E1 -27357.03,E2 -27357.03} C_VEL
LIN {X 0,Y 112.478,Z 447.374,A -85,B 0,C 180,E1 -27361.408,E2 -27361.408} C_VEL
LIN {X 0,Y 119.951,Z 444.501,A -85,B 0,C 180,E1 -27365.125,E2 -27365.125} C_VEL
LIN {X 0,Y 127.883,Z 440.311,A -85,B 0,C 180,E1 -27368.434,E2 -27368.434} C_VEL
LIN {X 0,Y 136.163,Z 434.67,A -85,B 0,C 180,E1 -27371.292,E2 -27371.292} C_VEL
LIN {X 0,Y 141.544,Z 430.329,A -85,B 0,C 180,E1 -27372.915,E2 -27372.915} C_VEL
LIN {X 0,Y 148.241,Z 423.881,A -85,B 0,C 180,E1 -27374.765,E2 -27374.765} C_VEL
LIN {X 0,Y 154.606,Z 416.561,A -85,B 0,C 180,E1 -27376.269,E2 -27376.269} C_VEL
LIN {X 0,Y 160.312,Z 408.635,A -85,B 0,C 180,E1 -27377.554,E2 -27377.554} C_VEL
LIN {X 0,Y 166.191,Z 398.615,A -85,B 0,C 180,E1 -27378.748,E2 -27378.748} C_VEL
LIN {X 0,Y 167.309,Z 396.233,A -85,B 0,C 180,E1 -27378.996,E2 -27378.996} C_VEL
LIN {X 0,Y 167.948,Z 394.783,A -85,B 0,C 180,E1 -27379.298,E2 -27379.298} C_VEL
LIN {X 0,Y 167.975,Z 393.843,A -85,B 0,C 180,E1 -27382.123,E2 -27382.123} C_VEL
LIN {X 0,Y 168.015,Z 393.871,A -85,B 0,C 180,E1 -27384.729,E2 -27384.729} C_VEL
LIN {X 0,Y 167.948,Z 395.115,A -85,B 0,C 180,E1 -27387.409,E2 -27387.409} C_VEL
LIN {X 0,Y 167.779,Z 396.06,A -85,B 0,C 180,E1 -27388.402,E2 -27388.402} C_VEL
LIN {X 0,Y 167.549,Z 396.795,A -85,B 0,C 180,E1 -27388.773,E2 -27388.773} C_VEL
LIN {X 0,Y 163.323,Z 405.01,A -85,B 0,C 180,E1 -27389.397,E2 -27389.397} C_VEL
LIN {X 0,Y 158.56,Z 412.713,A -85,B 0,C 180,E1 -27390.198,E2 -27390.198} C_VEL
LIN {X 0,Y 152.245,Z 421.22,A -85,B 0,C 180,E1 -27391.353,E2 -27391.353} C_VEL
LIN {X 0,Y 144.503,Z 429.786,A -85,B 0,C 180,E1 -27392.972,E2 -27392.972} C_VEL
LIN {X 0,Y 137.058,Z 436.508,A -85,B 0,C 180,E1 -27394.874,E2 -27394.874} C_VEL
LIN {X 0,Y 131.269,Z 441.02,A -85,B 0,C 180,E1 -27396.577,E2 -27396.577} C_VEL
LIN {X 0,Y 122.953,Z 446.426,A -85,B 0,C 180,E1 -27399.499,E2 -27399.499} C_VEL
LIN {X 0,Y 115.041,Z 450.543,A -85,B 0,C 180,E1 -27402.856,E2 -27402.856} C_VEL
LIN {X 0,Y 110.133,Z 452.626,A -85,B 0,C 180,E1 -27405.419,E2 -27405.419} C_VEL
LIN {X 0,Y 105.477,Z 454.269,A -85,B 0,C 180,E1 -27408.22,E2 -27408.22} C_VEL
LIN {X 0,Y 101.177,Z 455.368,A -85,B 0,C 180,E1 -27411.308,E2 -27411.308} C_VEL
LIN {X 0,Y 93.89,Z 456.254,A -85,B 0,C 180,E1 -27418.403,E2 -27418.403} C_VEL
LIN {X 0,Y 90.868,Z 456.098,A -85,B 0,C 180,E1 -27422.353,E2 -27422.353} C_VEL
LIN {X 0,Y 88.506,Z 455.405,A -85,B 0,C 180,E1 -27426.609,E2 -27426.609} C_VEL
LIN {X 0,Y 86.808,Z 454.316,A -85,B 0,C 180,E1 -27431.106,E2 -27431.106} C_VEL
LIN {X 0,Y 85.584,Z 452.802,A -85,B 0,C 180,E1 -27435.74,E2 -27435.74} C_VEL
LIN {X 0,Y 85.052,Z 449.702,A -85,B 0,C 180,E1 -27442.588,E2 -27442.588} C_VEL
LIN {X 0,Y 85.244,Z 446.712,A -85,B 0,C 180,E1 -27447.639,E2 -27447.639} C_VEL
LIN {X 0,Y 85.167,Z 441.94,A -85,B 0,C 180,E1 -27453.549,E2 -27453.549} C_VEL
LIN {X 0,Y 85.416,Z 435.771,A -85,B 0,C 180,E1 -27459.473,E2 -27459.473} C_VEL
LIN {X 0,Y 86.078,Z 429.67,A -85,B 0,C 180,E1 -27464.179,E2 -27464.179} C_VEL
LIN {X 0,Y 87.312,Z 422.275,A -85,B 0,C 180,E1 -27468.783,E2 -27468.783} C_VEL
LIN {X 0,Y 89.13,Z 413.158,A -85,B 0,C 180,E1 -27473.22,E2 -27473.22} C_VEL
LIN {X 0,Y 91.029,Z 402.659,A -85,B 0,C 180,E1 -27476.975,E2 -27476.975} C_VEL
LIN {X 0,Y 92.77,Z 393.036,A -85,B 0,C 180,E1 -27479.501,E2 -27479.501} C_VEL
LIN {X 0,Y 93.97,Z 384.047,A -85,B 0,C 180,E1 -27481.256,E2 -27481.256} C_VEL
LIN {X 0,Y 94.931,Z 374.39,A -85,B 0,C 180,E1 -27482.572,E2 -27482.572} C_VEL
LIN {X 0,Y 95.778,Z 359.92,A -85,B 0,C 180,E1 -27483.971,E2 -27483.971} C_VEL
LIN {X 0,Y 93.851,Z 325.087,A -85,B 0,C 180,E1 -27488.005,E2 -27488.005} C_VEL
LIN {X 0,Y 90.859,Z 314.889,A -85,B 0,C 180,E1 -27489.828,E2 -27489.828} C_VEL
LIN {X 0,Y 86.566,Z 304.886,A -85,B 0,C 180,E1 -27492.118,E2 -27492.118} C_VEL
LIN {X 0,Y 86.53,Z 304.512,A -85,B 0,C 180,E1 -27492.226,E2 -27492.226} C_VEL
LIN {X 0,Y 86.458,Z 304.524,A -85,B 0,C 180,E1 -27499.431,E2 -27499.431} C_VEL
LIN {X 0,Y 86.531,Z 304.519,A -85,B 0,C 180,E1 -27505.347,E2 -27505.347} C_VEL
LIN {X 0,Y 86.585,Z 304.511,A -85,B 0,C 180,E1 -27513.234,E2 -27513.234} C_VEL
LIN {X 0,Y 86.647,Z 304.502,A -85,B 0,C 180,E1 -27521.064,E2 -27521.064} C_VEL
LIN {X 0,Y 86.933,Z 304.462,A -85,B 0,C 180,E1 -27525.96,E2 -27525.96} C_VEL
LIN {X 0,Y 87.086,Z 304.449,A -85,B 0,C 180,E1 -27530.708,E2 -27530.708} C_VEL
LIN {X 0,Y 87.506,Z 304.388,A -85,B 0,C 180,E1 -27538.629,E2 -27538.629} C_VEL
LIN {X 0,Y 87.4,Z 304.41,A -85,B 0,C 180,E1 -27541.174,E2 -27541.174} C_VEL
LIN {X 0,Y 86.022,Z 304.587,A -85,B 0,C 180,E1 -27544.955,E2 -27544.955} C_VEL
LIN {X 0,Y 82.309,Z 305.042,A -85,B 0,C 180,E1 -27551.359,E2 -27551.359} C_VEL
LIN {X 0,Y 79.608,Z 305.379,A -85,B 0,C 180,E1 -27558.428,E2 -27558.428} C_VEL
LIN {X 0,Y 79.506,Z 305.381,A -85,B 0,C 180,E1 -27559.914,E2 -27559.914} C_VEL
LIN {X 0,Y 79.481,Z 305.391,A -85,B 0,C 180,E1 -27567.842,E2 -27567.842} C_VEL
LIN {X 0,Y 79.386,Z 305.407,A -85,B 0,C 180,E1 -27572.079,E2 -27572.079} C_VEL
LIN {X 0,Y 79.394,Z 305.4,A -85,B 0,C 180,E1 -27578.284,E2 -27578.284} C_VEL
LIN {X 0,Y 79.462,Z 305.393,A -85,B 0,C 180,E1 -27585.03,E2 -27585.03} C_VEL
LIN {X 0,Y 79.448,Z 305.398,A -85,B 0,C 180,E1 -27592.755,E2 -27592.755} C_VEL
LIN {X 0,Y 79.479,Z 305.391,A -85,B 0,C 180,E1 -27602.149,E2 -27602.149} C_VEL
LIN {X 0,Y 79.509,Z 305.391,A -85,B 0,C 180,E1 -27609.293,E2 -27609.293} C_VEL
LIN {X 0,Y 79.836,Z 305.353,A -85,B 0,C 180,E1 -27615.524,E2 -27615.524} C_VEL
LIN {X 0,Y 79.986,Z 305.326,A -85,B 0,C 180,E1 -27619.878,E2 -27619.878} C_VEL
LIN {X 0,Y 80.643,Z 305.246,A -85,B 0,C 180,E1 -27629.999,E2 -27629.999} C_VEL
LIN {X 0,Y 80.128,Z 305.31,A -85,B 0,C 180,E1 -27635.898,E2 -27635.898} C_VEL
LIN {X 0,Y 81.212,Z 308.331,A -85,B 0,C 180,E1 -27636.79,E2 -27636.79} C_VEL
LIN {X 0,Y 85.489,Z 319.446,A -85,B 0,C 180,E1 -27639.45,E2 -27639.45} C_VEL
LIN {X 0,Y 90.377,Z 334.118,A -85,B 0,C 180,E1 -27642.347,E2 -27642.347} C_VEL
LIN {X 0,Y 87.959,Z 367.599,A -85,B 0,C 180,E1 -27645.72,E2 -27645.72} C_VEL
LIN {X 0,Y 86.584,Z 378.92,A -85,B 0,C 180,E1 -27647.601,E2 -27647.601} C_VEL
LIN {X 0,Y 84.855,Z 390.093,A -85,B 0,C 180,E1 -27650.475,E2 -27650.475} C_VEL
LIN {X 0,Y 83.395,Z 397.961,A -85,B 0,C 180,E1 -27653.132,E2 -27653.132} C_VEL
LIN {X 0,Y 81.726,Z 405.458,A -85,B 0,C 180,E1 -27656.287,E2 -27656.287} C_VEL
LIN {X 0,Y 80.23,Z 412.916,A -85,B 0,C 180,E1 -27660.22,E2 -27660.22} C_VEL
LIN {X 0,Y 78.732,Z 420.697,A -85,B 0,C 180,E1 -27665.372,E2 -27665.372} C_VEL
LIN {X 0,Y 77.531,Z 427.721,A -85,B 0,C 180,E1 -27671.235,E2 -27671.235} C_VEL
LIN {X 0,Y 76.926,Z 434.603,A -85,B 0,C 180,E1 -27678.586,E2 -27678.586} C_VEL
LIN {X 0,Y 77.331,Z 439.239,A -85,B 0,C 180,E1 -27684.875,E2 -27684.875} C_VEL
LIN {X 0,Y 79.032,Z 443.8,A -85,B 0,C 180,E1 -27692.775,E2 -27692.775} C_VEL
LIN {X 0,Y 80.551,Z 445.809,A -85,B 0,C 180,E1 -27696.887,E2 -27696.887} C_VEL
LIN {X 0,Y 85.6,Z 448.886,A -85,B 0,C 180,E1 -27705.745,E2 -27705.745} C_VEL
LIN {X 0,Y 92.035,Z 450.222,A -85,B 0,C 180,E1 -27713.056,E2 -27713.056} C_VEL
LIN {X 0,Y 98.43,Z 450.128,A -85,B 0,C 180,E1 -27718.331,E2 -27718.331} C_VEL
LIN {X 0,Y 107.067,Z 448.454,A -85,B 0,C 180,E1 -27723.767,E2 -27723.767} C_VEL
LIN {X 0,Y 113.958,Z 446.235,A -85,B 0,C 180,E1 -27727.088,E2 -27727.088} C_VEL
LIN {X 0,Y 121.352,Z 443.009,A -85,B 0,C 180,E1 -27730.1,E2 -27730.1} C_VEL
LIN {X 0,Y 128.67,Z 438.936,A -85,B 0,C 180,E1 -27732.622,E2 -27732.622} C_VEL
LIN {X 0,Y 136.537,Z 433.524,A -85,B 0,C 180,E1 -27734.916,E2 -27734.916} C_VEL
LIN {X 0,Y 144.518,Z 426.751,A -85,B 0,C 180,E1 -27736.967,E2 -27736.967} C_VEL
LIN {X 0,Y 151.522,Z 419.414,A -85,B 0,C 180,E1 -27738.509,E2 -27738.509} C_VEL
LIN {X 0,Y 157.789,Z 411.443,A -85,B 0,C 180,E1 -27739.802,E2 -27739.802} C_VEL
LIN {X 0,Y 162.843,Z 403.688,A -85,B 0,C 180,E1 -27740.753,E2 -27740.753} C_VEL
LIN {X 0,Y 164.655,Z 400.594,A -85,B 0,C 180,E1 -27741.062,E2 -27741.062} C_VEL
LIN {X 0,Y 164.79,Z 400.172,A -85,B 0,C 180,E1 -27742.573,E2 -27742.573} C_VEL
LIN {X 0,Y 164.791,Z 400.524,A -85,B 0,C 180,E1 -27745.246,E2 -27745.246} C_VEL
LIN {X 0,Y 164.726,Z 401.032,A -85,B 0,C 180,E1 -27746.371,E2 -27746.371} C_VEL
LIN {X 0,Y 164.253,Z 401.94,A -85,B 0,C 180,E1 -27746.659,E2 -27746.659} C_VEL
LIN {X 0,Y 159.217,Z 410.232,A -85,B 0,C 180,E1 -27747.346,E2 -27747.346} C_VEL
LIN {X 0,Y 153.568,Z 417.981,A -85,B 0,C 180,E1 -27748.244,E2 -27748.244} C_VEL
LIN {X 0,Y 147.132,Z 425.375,A -85,B 0,C 180,E1 -27749.342,E2 -27749.342} C_VEL
LIN {X 0,Y 140.813,Z 431.578,A -85,B 0,C 180,E1 -27750.58,E2 -27750.58} C_VEL
LIN {X 0,Y 133.172,Z 437.927,A -85,B 0,C 180,E1 -27752.397,E2 -27752.397} C_VEL
LIN {X 0,Y 127.206,Z 442.11,A -85,B 0,C 180,E1 -27754.034,E2 -27754.034} C_VEL
LIN {X 0,Y 118.585,Z 447.175,A -85,B 0,C 180,E1 -27756.865,E2 -27756.865} C_VEL
LIN {X 0,Y 110.357,Z 450.995,A -85,B 0,C 180,E1 -27760.166,E2 -27760.166} C_VEL
LIN {X 0,Y 105.212,Z 452.825,A -85,B 0,C 180,E1 -27762.714,E2 -27762.714} C_VEL
LIN {X 0,Y 100.305,Z 454.228,A -85,B 0,C 180,E1 -27765.522,E2 -27765.522} C_VEL
LIN {X 0,Y 95.737,Z 455.229,A -85,B 0,C 180,E1 -27768.65,E2 -27768.65} C_VEL
LIN {X 0,Y 91.659,Z 455.722,A -85,B 0,C 180,E1 -27772.166,E2 -27772.166} C_VEL
LIN {X 0,Y 84.658,Z 455.388,A -85,B 0,C 180,E1 -27780.128,E2 -27780.128} C_VEL
LIN {X 0,Y 82.051,Z 454.644,A -85,B 0,C 180,E1 -27784.644,E2 -27784.644} C_VEL
LIN {X 0,Y 80.157,Z 453.361,A -85,B 0,C 180,E1 -27789.471,E2 -27789.471} C_VEL
LIN {X 0,Y 78.377,Z 450.663,A -85,B 0,C 180,E1 -27797.047,E2 -27797.047} C_VEL
LIN {X 0,Y 78.2,Z 446.824,A -85,B 0,C 180,E1 -27804.845,E2 -27804.845} C_VEL
LIN {X 0,Y 78.26,Z 443.33,A -85,B 0,C 180,E1 -27810.001,E2 -27810.001} C_VEL
LIN {X 0,Y 78.214,Z 437.306,A -85,B 0,C 180,E1 -27816.87,E2 -27816.87} C_VEL
LIN {X 0,Y 78.843,Z 430.506,A -85,B 0,C 180,E1 -27822.877,E2 -27822.877} C_VEL
LIN {X 0,Y 79.906,Z 423.335,A -85,B 0,C 180,E1 -27827.93,E2 -27827.93} C_VEL
LIN {X 0,Y 81.434,Z 415.771,A -85,B 0,C 180,E1 -27832.184,E2 -27832.184} C_VEL
LIN {X 0,Y 82.977,Z 407.821,A -85,B 0,C 180,E1 -27835.728,E2 -27835.728} C_VEL
LIN {X 0,Y 84.87,Z 397.949,A -85,B 0,C 180,E1 -27839.112,E2 -27839.112} C_VEL
LIN {X 0,Y 86.825,Z 386.174,A -85,B 0,C 180,E1 -27841.916,E2 -27841.916} C_VEL
LIN {X 0,Y 87.943,Z 376.296,A -85,B 0,C 180,E1 -27843.499,E2 -27843.499} C_VEL
LIN {X 0,Y 88.928,Z 359.887,A -85,B 0,C 180,E1 -27845.274,E2 -27845.274} C_VEL
LIN {X 0,Y 87.242,Z 326.709,A -85,B 0,C 180,E1 -27849.387,E2 -27849.387} C_VEL
LIN {X 0,Y 84.582,Z 317.538,A -85,B 0,C 180,E1 -27851.174,E2 -27851.174} C_VEL
LIN {X 0,Y 79.585,Z 306.299,A -85,B 0,C 180,E1 -27854.145,E2 -27854.145} C_VEL
LIN {X 0,Y 79.403,Z 305.401,A -85,B 0,C 180,E1 -27854.465,E2 -27854.465} C_VEL
LIN {X 0,Y 79.387,Z 305.403,A -85,B 0,C 180,E1 -27862.822,E2 -27862.822} C_VEL
LIN {X 0,Y 79.378,Z 305.406,A -85,B 0,C 180,E1 -27867.907,E2 -27867.907} C_VEL
LIN {X 0,Y 79.526,Z 305.392,A -85,B 0,C 180,E1 -27873.773,E2 -27873.773} C_VEL
LIN {X 0,Y 79.515,Z 305.385,A -85,B 0,C 180,E1 -27879.291,E2 -27879.291} C_VEL
LIN {X 0,Y 79.827,Z 305.348,A -85,B 0,C 180,E1 -27885.569,E2 -27885.569} C_VEL
LIN {X 0,Y 79.969,Z 305.335,A -85,B 0,C 180,E1 -27889.872,E2 -27889.872} C_VEL
LIN {X 0,Y 80.644,Z 305.252,A -85,B 0,C 180,E1 -27899.996,E2 -27899.996} C_VEL
LIN {X 0,Y 79.992,Z 305.33,A -85,B 0,C 180,E1 -27910.116,E2 -27910.116} C_VEL
LIN {X 0,Y 79.762,Z 305.361,A -85,B 0,C 180,E1 -27915.323,E2 -27915.323} C_VEL
LIN {X 0,Y 79.506,Z 305.381,A -85,B 0,C 180,E1 -27919.914,E2 -27919.914} C_VEL
LIN {X 0,Y 79.193,Z 305.432,A -85,B 0,C 180,E1 -27922.74,E2 -27922.74} C_VEL
LIN {X 0,Y 77.865,Z 305.614,A -85,B 0,C 180,E1 -27926.949,E2 -27926.949} C_VEL
LIN {X 0,Y 74.69,Z 306.019,A -85,B 0,C 180,E1 -27934.121,E2 -27934.121} C_VEL
LIN {X 0,Y 72.66,Z 306.258,A -85,B 0,C 180,E1 -27940.295,E2 -27940.295} C_VEL
LIN {X 0,Y 72.272,Z 306.29,A -85,B 0,C 180,E1 -27943.515,E2 -27943.515} C_VEL
LIN {X 0,Y 72.355,Z 306.285,A -85,B 0,C 180,E1 -27950.984,E2 -27950.984} C_VEL
LIN {X 0,Y 72.334,Z 306.278,A -85,B 0,C 180,E1 -27954.34,E2 -27954.34} C_VEL
LIN {X 0,Y 72.387,Z 306.278,A -85,B 0,C 180,E1 -27960.957,E2 -27960.957} C_VEL
LIN {X 0,Y 72.39,Z 306.28,A -85,B 0,C 180,E1 -27967.148,E2 -27967.148} C_VEL
LIN {X 0,Y 72.73,Z 306.237,A -85,B 0,C 180,E1 -27975.064,E2 -27975.064} C_VEL
LIN {X 0,Y 72.874,Z 306.214,A -85,B 0,C 180,E1 -27978.878,E2 -27978.878} C_VEL
LIN {X 0,Y 73.57,Z 306.127,A -85,B 0,C 180,E1 -27989.999,E2 -27989.999} C_VEL
LIN {X 0,Y 73.175,Z 306.183,A -85,B 0,C 180,E1 -27993.612,E2 -27993.612} C_VEL
LIN {X 0,Y 74.994,Z 311.1,A -85,B 0,C 180,E1 -27995.039,E2 -27995.039} C_VEL
LIN {X 0,Y 78.205,Z 319.134,A -85,B 0,C 180,E1 -27997.209,E2 -27997.209} C_VEL
LIN {X 0,Y 83.601,Z 335.286,A -85,B 0,C 180,E1 -28000.833,E2 -28000.833} C_VEL
LIN {X 0,Y 81.305,Z 366.529,A -85,B 0,C 180,E1 -28004.188,E2 -28004.188} C_VEL
LIN {X 0,Y 80.011,Z 377.028,A -85,B 0,C 180,E1 -28005.938,E2 -28005.938} C_VEL
LIN {X 0,Y 78.256,Z 388.389,A -85,B 0,C 180,E1 -28008.793,E2 -28008.793} C_VEL
LIN {X 0,Y 76.404,Z 397.874,A -85,B 0,C 180,E1 -28012.163,E2 -28012.163} C_VEL
LIN {X 0,Y 74.472,Z 406.391,A -85,B 0,C 180,E1 -28016.104,E2 -28016.104} C_VEL
LIN {X 0,Y 73.055,Z 413.136,A -85,B 0,C 180,E1 -28020.034,E2 -28020.034} C_VEL
LIN {X 0,Y 71.628,Z 420.433,A -85,B 0,C 180,E1 -28025.317,E2 -28025.317} C_VEL
LIN {X 0,Y 70.449,Z 427.141,A -85,B 0,C 180,E1 -28031.401,E2 -28031.401} C_VEL
LIN {X 0,Y 69.934,Z 432.423,A -85,B 0,C 180,E1 -28037.293,E2 -28037.293} C_VEL
LIN {X 0,Y 70.072,Z 436.949,A -85,B 0,C 180,E1 -28043.354,E2 -28043.354} C_VEL
LIN {X 0,Y 71.218,Z 441.352,A -85,B 0,C 180,E1 -28050.441,E2 -28050.441} C_VEL
LIN {X 0,Y 73.379,Z 444.91,A -85,B 0,C 180,E1 -28057.479,E2 -28057.479} C_VEL
LIN {X 0,Y 76.666,Z 447.577,A -85,B 0,C 180,E1 -28064.042,E2 -28064.042} C_VEL
LIN {X 0,Y 80.826,Z 449.407,A -85,B 0,C 180,E1 -28069.989,E2 -28069.989} C_VEL
LIN {X 0,Y 85.829,Z 450.451,A -85,B 0,C 180,E1 -28075.307,E2 -28075.307} C_VEL
LIN {X 0,Y 91.539,Z 450.707,A -85,B 0,C 180,E1 -28080.004,E2 -28080.004} C_VEL
LIN {X 0,Y 98.713,Z 450.035,A -85,B 0,C 180,E1 -28084.65,E2 -28084.65} C_VEL
LIN {X 0,Y 106.616,Z 448.305,A -85,B 0,C 180,E1 -28088.605,E2 -28088.605} C_VEL
LIN {X 0,Y 114.941,Z 445.484,A -85,B 0,C 180,E1 -28091.964,E2 -28091.964} C_VEL
LIN {X 0,Y 125.537,Z 440.282,A -85,B 0,C 180,E1 -28095.431,E2 -28095.431} C_VEL
LIN {X 0,Y 132.487,Z 435.947,A -85,B 0,C 180,E1 -28097.292,E2 -28097.292} C_VEL
LIN {X 0,Y 139.186,Z 430.947,A -85,B 0,C 180,E1 -28098.885,E2 -28098.885} C_VEL
LIN {X 0,Y 146.051,Z 424.802,A -85,B 0,C 180,E1 -28100.355,E2 -28100.355} C_VEL
LIN {X 0,Y 152.687,Z 417.664,A -85,B 0,C 180,E1 -28101.609,E2 -28101.609} C_VEL
LIN {X 0,Y 158.193,Z 410.569,A -85,B 0,C 180,E1 -28102.568,E2 -28102.568} C_VEL
LIN {X 0,Y 161.102,Z 406.335,A -85,B 0,C 180,E1 -28103.12,E2 -28103.12} C_VEL
LIN {X 0,Y 161.078,Z 406.389,A -85,B 0,C 180,E1 -28103.62,E2 -28103.62} C_VEL
LIN {X 0,Y 160.382,Z 407.695,A -85,B 0,C 180,E1 -28104.563,E2 -28104.563} C_VEL
LIN {X 0,Y 153.691,Z 416.908,A -85,B 0,C 180,E1 -28105.431,E2 -28105.431} C_VEL
LIN {X 0,Y 147.105,Z 424.4,A -85,B 0,C 180,E1 -28106.394,E2 -28106.394} C_VEL
LIN {X 0,Y 140.593,Z 430.653,A -85,B 0,C 180,E1 -28107.469,E2 -28107.469} C_VEL
LIN {X 0,Y 134.241,Z 435.885,A -85,B 0,C 180,E1 -28108.73,E2 -28108.73} C_VEL
LIN {X 0,Y 126.467,Z 441.285,A -85,B 0,C 180,E1 -28110.534,E2 -28110.534} C_VEL
LIN {X 0,Y 117.428,Z 446.433,A -85,B 0,C 180,E1 -28113.085,E2 -28113.085} C_VEL
LIN {X 0,Y 108.753,Z 450.308,A -85,B 0,C 180,E1 -28116.122,E2 -28116.122} C_VEL
LIN {X 0,Y 100.548,Z 453.035,A -85,B 0,C 180,E1 -28119.751,E2 -28119.751} C_VEL
LIN {X 0,Y 90.53,Z 454.949,A -85,B 0,C 180,E1 -28125.681,E2 -28125.681} C_VEL
LIN {X 0,Y 86.173,Z 455.344,A -85,B 0,C 180,E1 -28129.276,E2 -28129.276} C_VEL
LIN {X 0,Y 82.166,Z 455.229,A -85,B 0,C 180,E1 -28133.223,E2 -28133.223} C_VEL
LIN {X 0,Y 78.601,Z 454.643,A -85,B 0,C 180,E1 -28137.558,E2 -28137.558} C_VEL
LIN {X 0,Y 75.741,Z 453.71,A -85,B 0,C 180,E1 -28142.36,E2 -28142.36} C_VEL
LIN {X 0,Y 73.584,Z 452.374,A -85,B 0,C 180,E1 -28147.542,E2 -28147.542} C_VEL
LIN {X 0,Y 71.589,Z 449.363,A -85,B 0,C 180,E1 -28155.795,E2 -28155.795} C_VEL
LIN {X 0,Y 71.327,Z 445.199,A -85,B 0,C 180,E1 -28164.347,E2 -28164.347} C_VEL
LIN {X 0,Y 71.409,Z 443.499,A -85,B 0,C 180,E1 -28167.181,E2 -28167.181} C_VEL
LIN {X 0,Y 71.201,Z 438.191,A -85,B 0,C 180,E1 -28174.247,E2 -28174.247} C_VEL
LIN {X 0,Y 71.626,Z 431.329,A -85,B 0,C 180,E1 -28181.318,E2 -28181.318} C_VEL
LIN {X 0,Y 72.727,Z 423.413,A -85,B 0,C 180,E1 -28187.578,E2 -28187.578} C_VEL
LIN {X 0,Y 74.21,Z 415.927,A -85,B 0,C 180,E1 -28192.261,E2 -28192.261} C_VEL
LIN {X 0,Y 75.849,Z 408.141,A -85,B 0,C 180,E1 -28196.113,E2 -28196.113} C_VEL
LIN {X 0,Y 77.417,Z 400.176,A -85,B 0,C 180,E1 -28199.207,E2 -28199.207} C_VEL
LIN {X 0,Y 79.328,Z 390.194,A -85,B 0,C 180,E1 -28202.112,E2 -28202.112} C_VEL
LIN {X 0,Y 80.948,Z 377.96,A -85,B 0,C 180,E1 -28204.546,E2 -28204.546} C_VEL
LIN {X 0,Y 82.179,Z 360.714,A -85,B 0,C 180,E1 -28206.582,E2 -28206.582} C_VEL
LIN {X 0,Y 80.641,Z 327.981,A -85,B 0,C 180,E1 -28211.021,E2 -28211.021} C_VEL
LIN {X 0,Y 78.517,Z 320.585,A -85,B 0,C 180,E1 -28212.632,E2 -28212.632} C_VEL
LIN {X 0,Y 73.321,Z 309.157,A -85,B 0,C 180,E1 -28216.035,E2 -28216.035} C_VEL
LIN {X 0,Y 72.25,Z 306.298,A -85,B 0,C 180,E1 -28216.947,E2 -28216.947} C_VEL
LIN {X 0,Y 72.295,Z 306.291,A -85,B 0,C 180,E1 -28224.313,E2 -28224.313} C_VEL
LIN {X 0,Y 72.361,Z 306.277,A -85,B 0,C 180,E1 -28230.942,E2 -28230.942} C_VEL
LIN {X 0,Y 72.395,Z 306.273,A -85,B 0,C 180,E1 -28237.146,E2 -28237.146} C_VEL
LIN {X 0,Y 72.723,Z 306.234,A -85,B 0,C 180,E1 -28245.106,E2 -28245.106} C_VEL
LIN {X 0,Y 72.86,Z 306.218,A -85,B 0,C 180,E1 -28248.872,E2 -28248.872} C_VEL
LIN {X 0,Y 73.57,Z 306.133,A -85,B 0,C 180,E1 -28259.995,E2 -28259.995} C_VEL
LIN {X 0,Y 72.879,Z 306.213,A -85,B 0,C 180,E1 -28271.115,E2 -28271.115} C_VEL
LIN {X 0,Y 72.582,Z 306.256,A -85,B 0,C 180,E1 -28276.882,E2 -28276.882} C_VEL
LIN {X 0,Y 72.393,Z 306.276,A -85,B 0,C 180,E1 -28282.845,E2 -28282.845} C_VEL
LIN {X 0,Y 72.374,Z 306.274,A -85,B 0,C 180,E1 -28289.078,E2 -28289.078} C_VEL
LIN {X 0,Y 72.308,Z 306.287,A -85,B 0,C 180,E1 -28295.667,E2 -28295.667} C_VEL
LIN {X 0,Y 72.272,Z 306.29,A -85,B 0,C 180,E1 -28303.515,E2 -28303.515} C_VEL
LIN {X 0,Y 71.866,Z 306.337,A -85,B 0,C 180,E1 -28306.622,E2 -28306.622} C_VEL
LIN {X 0,Y 70.421,Z 306.526,A -85,B 0,C 180,E1 -28311.25,E2 -28311.25} C_VEL
LIN {X 0,Y 67.204,Z 306.927,A -85,B 0,C 180,E1 -28319.2,E2 -28319.2} C_VEL
LIN {X 0,Y 65.408,Z 307.148,A -85,B 0,C 180,E1 -28326.105,E2 -28326.105} C_VEL
LIN {X 0,Y 65.271,Z 307.149,A -85,B 0,C 180,E1 -28329.685,E2 -28329.685} C_VEL
LIN {X 0,Y 65.631,Z 307.121,A -85,B 0,C 180,E1 -28334.505,E2 -28334.505} C_VEL
LIN {X 0,Y 65.767,Z 307.103,A -85,B 0,C 180,E1 -28337.658,E2 -28337.658} C_VEL
LIN {X 0,Y 66.494,Z 307.008,A -85,B 0,C 180,E1 -28349.999,E2 -28349.999} C_VEL
LIN {X 0,Y 66.391,Z 307.023,A -85,B 0,C 180,E1 -28350.756,E2 -28350.756} C_VEL
LIN {X 0,Y 67.296,Z 309.855,A -85,B 0,C 180,E1 -28351.68,E2 -28351.68} C_VEL
LIN {X 0,Y 71.894,Z 321.244,A -85,B 0,C 180,E1 -28355.333,E2 -28355.333} C_VEL
LIN {X 0,Y 76.92,Z 336.674,A -85,B 0,C 180,E1 -28359.122,E2 -28359.122} C_VEL
LIN {X 0,Y 74.435,Z 367.654,A -85,B 0,C 180,E1 -28362.736,E2 -28362.736} C_VEL
LIN {X 0,Y 72.889,Z 379.011,A -85,B 0,C 180,E1 -28364.861,E2 -28364.861} C_VEL
LIN {X 0,Y 71.074,Z 389.75,A -85,B 0,C 180,E1 -28367.998,E2 -28367.998} C_VEL
LIN {X 0,Y 69.363,Z 398.044,A -85,B 0,C 180,E1 -28371.244,E2 -28371.244} C_VEL
LIN {X 0,Y 67.397,Z 406.406,A -85,B 0,C 180,E1 -28375.474,E2 -28375.474} C_VEL
LIN {X 0,Y 65.91,Z 413.079,A -85,B 0,C 180,E1 -28379.71,E2 -28379.71} C_VEL
LIN {X 0,Y 64.315,Z 421.021,A -85,B 0,C 180,E1 -28386.092,E2 -28386.092} C_VEL
LIN {X 0,Y 63.366,Z 426.658,A -85,B 0,C 180,E1 -28391.715,E2 -28391.715} C_VEL
LIN {X 0,Y 62.895,Z 431.818,A -85,B 0,C 180,E1 -28397.906,E2 -28397.906} C_VEL
LIN {X 0,Y 63.344,Z 437.528,A -85,B 0,C 180,E1 -28406.313,E2 -28406.313} C_VEL
LIN {X 0,Y 64.995,Z 442.018,A -85,B 0,C 180,E1 -28414.378,E2 -28414.378} C_VEL
LIN {X 0,Y 67.832,Z 445.518,A -85,B 0,C 180,E1 -28421.896,E2 -28421.896} C_VEL
LIN {X 0,Y 71.754,Z 448.139,A -85,B 0,C 180,E1 -28428.708,E2 -28428.708} C_VEL
LIN {X 0,Y 77.519,Z 450.192,A -85,B 0,C 180,E1 -28435.736,E2 -28435.736} C_VEL
LIN {X 0,Y 84.369,Z 451.159,A -85,B 0,C 180,E1 -28441.676,E2 -28441.676} C_VEL
LIN {X 0,Y 91.974,Z 451.051,A -85,B 0,C 180,E1 -28446.621,E2 -28446.621} C_VEL
LIN {X 0,Y 100.135,Z 449.847,A -85,B 0,C 180,E1 -28450.716,E2 -28450.716} C_VEL
LIN {X 0,Y 110.537,Z 446.893,A -85,B 0,C 180,E1 -28454.736,E2 -28454.736} C_VEL
LIN {X 0,Y 118.619,Z 443.648,A -85,B 0,C 180,E1 -28457.235,E2 -28457.235} C_VEL
LIN {X 0,Y 126.939,Z 439.335,A -85,B 0,C 180,E1 -28459.404,E2 -28459.404} C_VEL
LIN {X 0,Y 135.815,Z 433.557,A -85,B 0,C 180,E1 -28461.344,E2 -28461.344} C_VEL
LIN {X 0,Y 144.169,Z 426.638,A -85,B 0,C 180,E1 -28462.956,E2 -28462.956} C_VEL
LIN {X 0,Y 145.203,Z 425.631,A -85,B 0,C 180,E1 -28463.133,E2 -28463.133} C_VEL
LIN {X 0,Y 145.803,Z 425.105,A -85,B 0,C 180,E1 -28463.68,E2 -28463.68} C_VEL
LIN {X 0,Y 137.513,Z 432.582,A -85,B 0,C 180,E1 -28464.888,E2 -28464.888} C_VEL
LIN {X 0,Y 129.418,Z 438.575,A -85,B 0,C 180,E1 -28466.364,E2 -28466.364} C_VEL
LIN {X 0,Y 119.897,Z 444.196,A -85,B 0,C 180,E1 -28468.452,E2 -28468.452} C_VEL
LIN {X 0,Y 110.689,Z 448.445,A -85,B 0,C 180,E1 -28471.005,E2 -28471.005} C_VEL
LIN {X 0,Y 101.807,Z 451.571,A -85,B 0,C 180,E1 -28474.07,E2 -28474.07} C_VEL
LIN {X 0,Y 96.167,Z 453.078,A -85,B 0,C 180,E1 -28476.5,E2 -28476.5} C_VEL
LIN {X 0,Y 90.744,Z 454.153,A -85,B 0,C 180,E1 -28479.245,E2 -28479.245} C_VEL
LIN {X 0,Y 85.598,Z 454.676,A -85,B 0,C 180,E1 -28482.362,E2 -28482.362} C_VEL
LIN {X 0,Y 76.616,Z 454.61,A -85,B 0,C 180,E1 -28490.053,E2 -28490.053} C_VEL
LIN {X 0,Y 72.73,Z 453.891,A -85,B 0,C 180,E1 -28494.567,E2 -28494.567} C_VEL
LIN {X 0,Y 67.148,Z 451.179,A -85,B 0,C 180,E1 -28505.252,E2 -28505.252} C_VEL
LIN {X 0,Y 64.86,Z 447.944,A -85,B 0,C 180,E1 -28514.285,E2 -28514.285} C_VEL
LIN {X 0,Y 64.402,Z 444.548,A -85,B 0,C 180,E1 -28521.79,E2 -28521.79} C_VEL
LIN {X 0,Y 64.493,Z 441.783,A -85,B 0,C 180,E1 -28526.878,E2 -28526.878} C_VEL
LIN {X 0,Y 64.264,Z 436.05,A -85,B 0,C 180,E1 -28534.706,E2 -28534.706} C_VEL
LIN {X 0,Y 64.8,Z 428.702,A -85,B 0,C 180,E1 -28542.529,E2 -28542.529} C_VEL
LIN {X 0,Y 65.89,Z 421.389,A -85,B 0,C 180,E1 -28548.663,E2 -28548.663} C_VEL
LIN {X 0,Y 67.574,Z 413.675,A -85,B 0,C 180,E1 -28553.768,E2 -28553.768} C_VEL
LIN {X 0,Y 69.607,Z 404.049,A -85,B 0,C 180,E1 -28558.66,E2 -28558.66} C_VEL
LIN {X 0,Y 71.862,Z 393.067,A -85,B 0,C 180,E1 -28562.541,E2 -28562.541} C_VEL
LIN {X 0,Y 73.356,Z 383.835,A -85,B 0,C 180,E1 -28564.88,E2 -28564.88} C_VEL
LIN {X 0,Y 74.464,Z 374.733,A -85,B 0,C 180,E1 -28566.498,E2 -28566.498} C_VEL
LIN {X 0,Y 75.411,Z 360.952,A -85,B 0,C 180,E1 -28568.225,E2 -28568.225} C_VEL
LIN {X 0,Y 74.134,Z 329.502,A -85,B 0,C 180,E1 -28572.892,E2 -28572.892} C_VEL
LIN {X 0,Y 72.284,Z 323.151,A -85,B 0,C 180,E1 -28574.418,E2 -28574.418} C_VEL
LIN {X 0,Y 67.571,Z 312.707,A -85,B 0,C 180,E1 -28577.884,E2 -28577.884} C_VEL
LIN {X 0,Y 65.395,Z 308.164,A -85,B 0,C 180,E1 -28579.644,E2 -28579.644} C_VEL
LIN {X 0,Y 65.218,Z 307.168,A -85,B 0,C 180,E1 -28579.963,E2 -28579.963} C_VEL
LIN {X 0,Y 65.172,Z 307.177,A -85,B 0,C 180,E1 -28587.366,E2 -28587.366} C_VEL
LIN {X 0,Y 65.234,Z 307.172,A -85,B 0,C 180,E1 -28594.467,E2 -28594.467} C_VEL
LIN {X 0,Y 65.62,Z 307.121,A -85,B 0,C 180,E1 -28604.563,E2 -28604.563} C_VEL
LIN {X 0,Y 65.757,Z 307.098,A -85,B 0,C 180,E1 -28607.652,E2 -28607.652} C_VEL
LIN {X 0,Y 66.493,Z 307.015,A -85,B 0,C 180,E1 -28619.995,E2 -28619.995} C_VEL
LIN {X 0,Y 65.772,Z 307.096,A -85,B 0,C 180,E1 -28632.334,E2 -28632.334} C_VEL
LIN {X 0,Y 65.385,Z 307.148,A -85,B 0,C 180,E1 -28638.806,E2 -28638.806} C_VEL
LIN {X 0,Y 65.246,Z 307.171,A -85,B 0,C 180,E1 -28645.516,E2 -28645.516} C_VEL
LIN {X 0,Y 65.201,Z 307.176,A -85,B 0,C 180,E1 -28652.606,E2 -28652.606} C_VEL
LIN {X 0,Y 65.222,Z 307.172,A -85,B 0,C 180,E1 -28661.036,E2 -28661.036} C_VEL
LIN {X 0,Y 65.263,Z 307.168,A -85,B 0,C 180,E1 -28669.749,E2 -28669.749} C_VEL
LIN {X 0,Y 65.255,Z 307.169,A -85,B 0,C 180,E1 -28679.485,E2 -28679.485} C_VEL
LIN {X 0,Y 65.241,Z 307.164,A -85,B 0,C 180,E1 -28684.475,E2 -28684.475} C_VEL
LIN {X 0,Y 65.271,Z 307.149,A -85,B 0,C 180,E1 -28689.685,E2 -28689.685} C_VEL
LIN {X 0,Y 64.667,Z 307.235,A -85,B 0,C 180,E1 -28691.717,E2 -28691.717} C_VEL
LIN {X 0,Y 62.021,Z 307.571,A -85,B 0,C 180,E1 -28694.655,E2 -28694.655} C_VEL
LIN {X 0,Y 59.268,Z 307.912,A -85,B 0,C 180,E1 -28697.848,E2 -28697.848} C_VEL
LIN {X 0,Y 58.633,Z 307.98,A -85,B 0,C 180,E1 -28700.213,E2 -28700.213} C_VEL
LIN {X 0,Y 59.083,Z 308.112,A -85,B 0,C 180,E1 -28707.015,E2 -28707.015} C_VEL
LIN {X 0,Y 60.238,Z 310.842,A -85,B 0,C 180,E1 -28708.199,E2 -28708.199} C_VEL
LIN {X 0,Y 61.606,Z 313.233,A -85,B 0,C 180,E1 -28709.378,E2 -28709.378} C_VEL
LIN {X 0,Y 65.986,Z 324.515,A -85,B 0,C 180,E1 -28713.43,E2 -28713.43} C_VEL
LIN {X 0,Y 70.223,Z 337.947,A -85,B 0,C 180,E1 -28717.161,E2 -28717.161} C_VEL
LIN {X 0,Y 67.658,Z 367.868,A -85,B 0,C 180,E1 -28720.925,E2 -28720.925} C_VEL
LIN {X 0,Y 66.148,Z 378.728,A -85,B 0,C 180,E1 -28723.109,E2 -28723.109} C_VEL
LIN {X 0,Y 64.065,Z 390.285,A -85,B 0,C 180,E1 -28726.74,E2 -28726.74} C_VEL
LIN {X 0,Y 62.175,Z 398.701,A -85,B 0,C 180,E1 -28730.38,E2 -28730.38} C_VEL
LIN {X 0,Y 60.095,Z 407.26,A -85,B 0,C 180,E1 -28735.244,E2 -28735.244} C_VEL
LIN {X 0,Y 58.285,Z 415.277,A -85,B 0,C 180,E1 -28741.171,E2 -28741.171} C_VEL
LIN {X 0,Y 56.984,Z 421.713,A -85,B 0,C 180,E1 -28747.196,E2 -28747.196} C_VEL
LIN {X 0,Y 55.983,Z 428.839,A -85,B 0,C 180,E1 -28755.605,E2 -28755.605} C_VEL
LIN {X 0,Y 56.194,Z 435.69,A -85,B 0,C 180,E1 -28765.763,E2 -28765.763} C_VEL
LIN {X 0,Y 58.448,Z 441.659,A -85,B 0,C 180,E1 -28777.003,E2 -28777.003} C_VEL
LIN {X 0,Y 62.695,Z 446.112,A -85,B 0,C 180,E1 -28787.05,E2 -28787.05} C_VEL
LIN {X 0,Y 67.356,Z 448.676,A -85,B 0,C 180,E1 -28794.016,E2 -28794.016} C_VEL
LIN {X 0,Y 72.895,Z 450.433,A -85,B 0,C 180,E1 -28800.005,E2 -28800.005} C_VEL
LIN {X 0,Y 79.233,Z 451.42,A -85,B 0,C 180,E1 -28805.093,E2 -28805.093} C_VEL
LIN {X 0,Y 86.153,Z 451.621,A -85,B 0,C 180,E1 -28809.394,E2 -28809.394} C_VEL
LIN {X 0,Y 93.818,Z 450.992,A -85,B 0,C 180,E1 -28813.144,E2 -28813.144} C_VEL
LIN {X 0,Y 106.088,Z 448.456,A -85,B 0,C 180,E1 -28817.628,E2 -28817.628} C_VEL
LIN {X 0,Y 114.857,Z 445.393,A -85,B 0,C 180,E1 -28820.114,E2 -28820.114} C_VEL
LIN {X 0,Y 123.861,Z 441.171,A -85,B 0,C 180,E1 -28822.225,E2 -28822.225} C_VEL
LIN {X 0,Y 126.787,Z 439.573,A -85,B 0,C 180,E1 -28822.834,E2 -28822.834} C_VEL
LIN {X 0,Y 125.231,Z 440.551,A -85,B 0,C 180,E1 -28823.725,E2 -28823.725} C_VEL
LIN {X 0,Y 116.7,Z 445.07,A -85,B 0,C 180,E1 -28825.403,E2 -28825.403} C_VEL
LIN {X 0,Y 107.224,Z 449.015,A -85,B 0,C 180,E1 -28827.77,E2 -28827.77} C_VEL
LIN {X 0,Y 98.015,Z 451.831,A -85,B 0,C 180,E1 -28830.638,E2 -28830.638} C_VEL
LIN {X 0,Y 86.44,Z 453.921,A -85,B 0,C 180,E1 -28835.609,E2 -28835.609} C_VEL
LIN {X 0,Y 80.99,Z 454.379,A -85,B 0,C 180,E1 -28838.652,E2 -28838.652} C_VEL
LIN {X 0,Y 71.338,Z 453.844,A -85,B 0,C 180,E1 -28846.403,E2 -28846.403} C_VEL
LIN {X 0,Y 67.103,Z 453.021,A -85,B 0,C 180,E1 -28851.07,E2 -28851.07} C_VEL
LIN {X 0,Y 63.587,Z 451.727,A -85,B 0,C 180,E1 -28856.455,E2 -28856.455} C_VEL
LIN {X 0,Y 59.736,Z 448.972,A -85,B 0,C 180,E1 -28865.686,E2 -28865.686} C_VEL
LIN {X 0,Y 57.736,Z 444.666,A -85,B 0,C 180,E1 -28876.884,E2 -28876.884} C_VEL
LIN {X 0,Y 57.62,Z 440.91,A -85,B 0,C 180,E1 -28884.753,E2 -28884.753} C_VEL
LIN {X 0,Y 57.36,Z 436.469,A -85,B 0,C 180,E1 -28891.757,E2 -28891.757} C_VEL
LIN {X 0,Y 57.596,Z 429.338,A -85,B 0,C 180,E1 -28900.551,E2 -28900.551} C_VEL
LIN {X 0,Y 58.559,Z 422.268,A -85,B 0,C 180,E1 -28907.458,E2 -28907.458} C_VEL
LIN {X 0,Y 60.141,Z 414.793,A -85,B 0,C 180,E1 -28913.23,E2 -28913.23} C_VEL
LIN {X 0,Y 61.879,Z 406.976,A -85,B 0,C 180,E1 -28917.938,E2 -28917.938} C_VEL
LIN {X 0,Y 63.985,Z 397.233,A -85,B 0,C 180,E1 -28922.376,E2 -28922.376} C_VEL
LIN {X 0,Y 66.126,Z 386.624,A -85,B 0,C 180,E1 -28925.773,E2 -28925.773} C_VEL
LIN {X 0,Y 67.607,Z 375.42,A -85,B 0,C 180,E1 -28928.115,E2 -28928.115} C_VEL
LIN {X 0,Y 68.704,Z 360.389,A -85,B 0,C 180,E1 -28930.202,E2 -28930.202} C_VEL
LIN {X 0,Y 67.71,Z 331.115,A -85,B 0,C 180,E1 -28934.955,E2 -28934.955} C_VEL
LIN {X 0,Y 66.08,Z 325.682,A -85,B 0,C 180,E1 -28936.477,E2 -28936.477} C_VEL
LIN {X 0,Y 61.766,Z 315.942,A -85,B 0,C 180,E1 -28940.199,E2 -28940.199} C_VEL
LIN {X 0,Y 59.086,Z 310.68,A -85,B 0,C 180,E1 -28942.701,E2 -28942.701} C_VEL
LIN {X 0,Y 58.186,Z 308.046,A -85,B 0,C 180,E1 -28943.923,E2 -28943.923} C_VEL
LIN {X 0,Y 58.133,Z 308.048,A -85,B 0,C 180,E1 -28951.074,E2 -28951.074} C_VEL
LIN {X 0,Y 58.513,Z 308.007,A -85,B 0,C 180,E1 -28963.922,E2 -28963.922} C_VEL
LIN {X 0,Y 58.8,Z 307.969,A -85,B 0,C 180,E1 -28973.13,E2 -28973.13} C_VEL
LIN {X 0,Y 59.384,Z 307.9,A -85,B 0,C 180,E1 -28979.994,E2 -28979.994} C_VEL
LIN {X 0,Y 58.816,Z 307.97,A -85,B 0,C 180,E1 -28986.857,E2 -28986.857} C_VEL
LIN {X 0,Y 58.525,Z 308.008,A -85,B 0,C 180,E1 -28996.117,E2 -28996.117} C_VEL
LIN {X 0,Y 58.152,Z 308.045,A -85,B 0,C 180,E1 -29008.902,E2 -29008.902} C_VEL
LIN {X 0,Y 58.052,Z 308.057,A -85,B 0,C 180,E1 -29017.244,E2 -29017.244} C_VEL
LIN {X 0,Y 58.084,Z 308.053,A -85,B 0,C 180,E1 -29026.541,E2 -29026.541} C_VEL
LIN {X 0,Y 58.07,Z 308.059,A -85,B 0,C 180,E1 -29032.761,E2 -29032.761} C_VEL
LIN {X 0,Y 58.152,Z 308.049,A -85,B 0,C 180,E1 -29041.089,E2 -29041.089} C_VEL
LIN {X 0,Y 58.52,Z 308.004,A -85,B 0,C 180,E1 -29053.874,E2 -29053.874} C_VEL
LIN {X 0,Y 58.633,Z 307.98,A -85,B 0,C 180,E1 -29060.213,E2 -29060.213} C_VEL
LIN {X 0,Y 58.646,Z 308.829,A -85,B 0,C 180,E1 -29062.769,E2 -29062.769} C_VEL
LIN {X 0,Y 58.545,Z 311.298,A -85,B 0,C 180,E1 -29065.231,E2 -29065.231} C_VEL
LIN {X 0,Y 58.415,Z 314.828,A -85,B 0,C 180,E1 -29067.094,E2 -29067.094} C_VEL
LIN {X 0,Y 58.643,Z 322.115,A -85,B 0,C 180,E1 -29069.333,E2 -29069.333} C_VEL
LIN {X 0,Y 59.708,Z 326.291,A -85,B 0,C 180,E1 -29070.713,E2 -29070.713} C_VEL
LIN {X 0,Y 63.751,Z 339.409,A -85,B 0,C 180,E1 -29074.875,E2 -29074.875} C_VEL
LIN {X 0,Y 60.975,Z 368.31,A -85,B 0,C 180,E1 -29078.768,E2 -29078.768} C_VEL
LIN {X 0,Y 59.239,Z 379.752,A -85,B 0,C 180,E1 -29081.279,E2 -29081.279} C_VEL
LIN {X 0,Y 57.127,Z 390.711,A -85,B 0,C 180,E1 -29085.153,E2 -29085.153} C_VEL
LIN {X 0,Y 55.035,Z 399.123,A -85,B 0,C 180,E1 -29089.212,E2 -29089.212} C_VEL
LIN {X 0,Y 52.965,Z 407.326,A -85,B 0,C 180,E1 -29094.47,E2 -29094.47} C_VEL
LIN {X 0,Y 51.16,Z 414.982,A -85,B 0,C 180,E1 -29100.855,E2 -29100.855} C_VEL
LIN {X 0,Y 49.823,Z 421.496,A -85,B 0,C 180,E1 -29107.728,E2 -29107.728} C_VEL
LIN {X 0,Y 49.002,Z 427.666,A -85,B 0,C 180,E1 -29115.813,E2 -29115.813} C_VEL
LIN {X 0,Y 49.119,Z 433.477,A -85,B 0,C 180,E1 -29125.097,E2 -29125.097} C_VEL
LIN {X 0,Y 50.735,Z 438.954,A -85,B 0,C 180,E1 -29135.452,E2 -29135.452} C_VEL
LIN {X 0,Y 53.798,Z 443.264,A -85,B 0,C 180,E1 -29144.861,E2 -29144.861} C_VEL
LIN {X 0,Y 58.174,Z 446.646,A -85,B 0,C 180,E1 -29153.067,E2 -29153.067} C_VEL
LIN {X 0,Y 63.614,Z 449.186,A -85,B 0,C 180,E1 -29160.005,E2 -29160.005} C_VEL
LIN {X 0,Y 70.715,Z 451.104,A -85,B 0,C 180,E1 -29166.38,E2 -29166.38} C_VEL
LIN {X 0,Y 78.942,Z 452.074,A -85,B 0,C 180,E1 -29171.691,E2 -29171.691} C_VEL
LIN {X 0,Y 87.685,Z 452.002,A -85,B 0,C 180,E1 -29175.894,E2 -29175.894} C_VEL
LIN {X 0,Y 96.733,Z 450.886,A -85,B 0,C 180,E1 -29179.185,E2 -29179.185} C_VEL
LIN {X 0,Y 106.01,Z 448.703,A -85,B 0,C 180,E1 -29181.859,E2 -29181.859} C_VEL
LIN {X 0,Y 109.331,Z 447.636,A -85,B 0,C 180,E1 -29182.69,E2 -29182.69} C_VEL
LIN {X 0,Y 107.343,Z 448.409,A -85,B 0,C 180,E1 -29183.569,E2 -29183.569} C_VEL
LIN {X 0,Y 100.926,Z 450.407,A -85,B 0,C 180,E1 -29185.147,E2 -29185.147} C_VEL
LIN {X 0,Y 94.603,Z 451.986,A -85,B 0,C 180,E1 -29186.946,E2 -29186.946} C_VEL
LIN {X 0,Y 88.47,Z 453.074,A -85,B 0,C 180,E1 -29189.097,E2 -29189.097} C_VEL
LIN {X 0,Y 76.763,Z 453.882,A -85,B 0,C 180,E1 -29194.517,E2 -29194.517} C_VEL
LIN {X 0,Y 71.432,Z 453.749,A -85,B 0,C 180,E1 -29198.088,E2 -29198.088} C_VEL
LIN {X 0,Y 61.799,Z 451.992,A -85,B 0,C 180,E1 -29206.977,E2 -29206.977} C_VEL
LIN {X 0,Y 57.861,Z 450.57,A -85,B 0,C 180,E1 -29212.608,E2 -29212.608} C_VEL
LIN {X 0,Y 53.472,Z 447.522,A -85,B 0,C 180,E1 -29222.614,E2 -29222.614} C_VEL
LIN {X 0,Y 51.146,Z 443.307,A -85,B 0,C 180,E1 -29234.15,E2 -29234.15} C_VEL
LIN {X 0,Y 50.834,Z 438.881,A -85,B 0,C 180,E1 -29244.05,E2 -29244.05} C_VEL
LIN {X 0,Y 50.452,Z 434.144,A -85,B 0,C 180,E1 -29251.998,E2 -29251.998} C_VEL
LIN {X 0,Y 50.606,Z 428.3,A -85,B 0,C 180,E1 -29260.001,E2 -29260.001} C_VEL
LIN {X 0,Y 51.537,Z 421.348,A -85,B 0,C 180,E1 -29267.663,E2 -29267.663} C_VEL
LIN {X 0,Y 53.24,Z 413.542,A -85,B 0,C 180,E1 -29274.365,E2 -29274.365} C_VEL
LIN {X 0,Y 55.424,Z 404.101,A -85,B 0,C 180,E1 -29280.48,E2 -29280.48} C_VEL
LIN {X 0,Y 58.111,Z 392.529,A -85,B 0,C 180,E1 -29285.595,E2 -29285.595} C_VEL
LIN {X 0,Y 59.768,Z 383.441,A -85,B 0,C 180,E1 -29288.391,E2 -29288.391} C_VEL
LIN {X 0,Y 61.039,Z 374.209,A -85,B 0,C 180,E1 -29290.367,E2 -29290.367} C_VEL
LIN {X 0,Y 62.081,Z 360.274,A -85,B 0,C 180,E1 -29292.475,E2 -29292.475} C_VEL
LIN {X 0,Y 61.245,Z 332.245,A -85,B 0,C 180,E1 -29297.603,E2 -29297.603} C_VEL
LIN {X 0,Y 59.484,Z 326.9,A -85,B 0,C 180,E1 -29299.465,E2 -29299.465} C_VEL
LIN {X 0,Y 55.49,Z 318.008,A -85,B 0,C 180,E1 -29303.492,E2 -29303.492} C_VEL
LIN {X 0,Y 52.736,Z 312.682,A -85,B 0,C 180,E1 -29306.546,E2 -29306.546} C_VEL
LIN {X 0,Y 51.209,Z 309.677,A -85,B 0,C 180,E1 -29308.443,E2 -29308.443} C_VEL
LIN {X 0,Y 51.082,Z 308.926,A -85,B 0,C 180,E1 -29308.932,E2 -29308.932} C_VEL
LIN {X 0,Y 51.389,Z 308.896,A -85,B 0,C 180,E1 -29323.203,E2 -29323.203} C_VEL
LIN {X 0,Y 51.676,Z 308.86,A -85,B 0,C 180,E1 -29332.177,E2 -29332.177} C_VEL
LIN {X 0,Y 52.267,Z 308.787,A -85,B 0,C 180,E1 -29339.993,E2 -29339.993} C_VEL
LIN {X 0,Y 51.691,Z 308.859,A -85,B 0,C 180,E1 -29347.807,E2 -29347.807} C_VEL
LIN {X 0,Y 51.393,Z 308.896,A -85,B 0,C 180,E1 -29356.811,E2 -29356.811} C_VEL
LIN {X 0,Y 51.026,Z 308.941,A -85,B 0,C 180,E1 -29364.399,E2 -29364.399} C_VEL
LIN {X 0,Y 51.037,Z 308.94,A -85,B 0,C 180,E1 -29374.286,E2 -29374.286} C_VEL
LIN {X 0,Y 51.042,Z 308.937,A -85,B 0,C 180,E1 -29383.498,E2 -29383.498} C_VEL
LIN {X 0,Y 51.048,Z 308.929,A -85,B 0,C 180,E1 -29386.497,E2 -29386.497} C_VEL
LIN {X 0,Y 51.07,Z 308.93,A -85,B 0,C 180,E1 -29396.6,E2 -29396.6} C_VEL
LIN {X 0,Y 51.023,Z 308.938,A -85,B 0,C 180,E1 -29405.591,E2 -29405.591} C_VEL
LIN {X 0,Y 51.461,Z 308.884,A -85,B 0,C 180,E1 -29414.147,E2 -29414.147} C_VEL
LIN {X 0,Y 51.698,Z 308.968,A -85,B 0,C 180,E1 -29421.939,E2 -29421.939} C_VEL
LIN {X 0,Y 52.709,Z 311.609,A -85,B 0,C 180,E1 -29423.351,E2 -29423.351} C_VEL
LIN {X 0,Y 54.59,Z 314.262,A -85,B 0,C 180,E1 -29425.309,E2 -29425.309} C_VEL
LIN {X 0,Y 56.29,Z 317.487,A -85,B 0,C 180,E1 -29427.096,E2 -29427.096} C_VEL
LIN {X 0,Y 59.708,Z 326.291,A -85,B 0,C 180,E1 -29430.713,E2 -29430.713} C_VEL
LIN {X 0,Y 60.648,Z 329.881,A -85,B 0,C 180,E1 -29431.82,E2 -29431.82} C_VEL
LIN {X 0,Y 60.812,Z 333.708,A -85,B 0,C 180,E1 -29432.567,E2 -29432.567} C_VEL
LIN {X 0,Y 60.388,Z 337.637,A -85,B 0,C 180,E1 -29433.057,E2 -29433.057} C_VEL
LIN {X 0,Y 56.259,Z 353.643,A -85,B 0,C 180,E1 -29434.021,E2 -29434.021} C_VEL
LIN {X 0,Y 55.55,Z 357.738,A -85,B 0,C 180,E1 -29434.455,E2 -29434.455} C_VEL
LIN {X 0,Y 53.811,Z 372.606,A -85,B 0,C 180,E1 -29436.959,E2 -29436.959} C_VEL
LIN {X 0,Y 51.687,Z 384.17,A -85,B 0,C 180,E1 -29440.414,E2 -29440.414} C_VEL
LIN {X 0,Y 49.649,Z 393.301,A -85,B 0,C 180,E1 -29444.375,E2 -29444.375} C_VEL
LIN {X 0,Y 47.29,Z 401.782,A -85,B 0,C 180,E1 -29449.325,E2 -29449.325} C_VEL
LIN {X 0,Y 45.076,Z 410.445,A -85,B 0,C 180,E1 -29456.224,E2 -29456.224} C_VEL
LIN {X 0,Y 42.837,Z 420.399,A -85,B 0,C 180,E1 -29467.21,E2 -29467.21} C_VEL
LIN {X 0,Y 41.968,Z 427.575,A -85,B 0,C 180,E1 -29477.956,E2 -29477.956} C_VEL
LIN {X 0,Y 42.624,Z 434.202,A -85,B 0,C 180,E1 -29490.363,E2 -29490.363} C_VEL
LIN {X 0,Y 45.066,Z 439.534,A -85,B 0,C 180,E1 -29501.834,E2 -29501.834} C_VEL
LIN {X 0,Y 49.594,Z 444.227,A -85,B 0,C 180,E1 -29512.71,E2 -29512.71} C_VEL
LIN {X 0,Y 56.263,Z 448.115,A -85,B 0,C 180,E1 -29522.215,E2 -29522.215} C_VEL
LIN {X 0,Y 64.117,Z 450.695,A -85,B 0,C 180,E1 -29529.44,E2 -29529.44} C_VEL
LIN {X 0,Y 75.349,Z 452.371,A -85,B 0,C 180,E1 -29536.254,E2 -29536.254} C_VEL
LIN {X 0,Y 83.417,Z 452.55,A -85,B 0,C 180,E1 -29539.699,E2 -29539.699} C_VEL
LIN {X 0,Y 91.886,Z 451.912,A -85,B 0,C 180,E1 -29542.488,E2 -29542.488} C_VEL
LIN {X 0,Y 91.606,Z 451.999,A -85,B 0,C 180,E1 -29542.986,E2 -29542.986} C_VEL
LIN {X 0,Y 85.25,Z 452.913,A -85,B 0,C 180,E1 -29544.933,E2 -29544.933} C_VEL
LIN {X 0,Y 79.042,Z 453.398,A -85,B 0,C 180,E1 -29547.239,E2 -29547.239} C_VEL
LIN {X 0,Y 72.982,Z 453.353,A -85,B 0,C 180,E1 -29549.93,E2 -29549.93} C_VEL
LIN {X 0,Y 61.873,Z 452.248,A -85,B 0,C 180,E1 -29557.338,E2 -29557.338} C_VEL
LIN {X 0,Y 56.865,Z 450.967,A -85,B 0,C 180,E1 -29562.141,E2 -29562.141} C_VEL
LIN {X 0,Y 48.891,Z 447.232,A -85,B 0,C 180,E1 -29574.904,E2 -29574.904} C_VEL
LIN {X 0,Y 45.206,Z 443.173,A -85,B 0,C 180,E1 -29587.136,E2 -29587.136} C_VEL
LIN {X 0,Y 44.158,Z 439.165,A -85,B 0,C 180,E1 -29597.82,E2 -29597.82} C_VEL
LIN {X 0,Y 44.041,Z 436.836,A -85,B 0,C 180,E1 -29603.129,E2 -29603.129} C_VEL
LIN {X 0,Y 43.524,Z 431.727,A -85,B 0,C 180,E1 -29612.316,E2 -29612.316} C_VEL
LIN {X 0,Y 44.11,Z 422.959,A -85,B 0,C 180,E1 -29624.822,E2 -29624.822} C_VEL
LIN {X 0,Y 45.808,Z 414.48,A -85,B 0,C 180,E1 -29633.748,E2 -29633.748} C_VEL
LIN {X 0,Y 47.686,Z 406.842,A -85,B 0,C 180,E1 -29639.83,E2 -29639.83} C_VEL
LIN {X 0,Y 49.606,Z 399.083,A -85,B 0,C 180,E1 -29644.522,E2 -29644.522} C_VEL
LIN {X 0,Y 52.182,Z 388.328,A -85,B 0,C 180,E1 -29649.149,E2 -29649.149} C_VEL
LIN {X 0,Y 54.181,Z 376.35,A -85,B 0,C 180,E1 -29652.507,E2 -29652.507} C_VEL
LIN {X 0,Y 55.567,Z 361.063,A -85,B 0,C 180,E1 -29655.11,E2 -29655.11} C_VEL
LIN {X 0,Y 55.064,Z 334.083,A -85,B 0,C 180,E1 -29660.553,E2 -29660.553} C_VEL
LIN {X 0,Y 52.188,Z 326.205,A -85,B 0,C 180,E1 -29664.002,E2 -29664.002} C_VEL
LIN {X 0,Y 47.984,Z 317.325,A -85,B 0,C 180,E1 -29669.458,E2 -29669.458} C_VEL
LIN {X 0,Y 46.122,Z 314.035,A -85,B 0,C 180,E1 -29672.175,E2 -29672.175} C_VEL
LIN {X 0,Y 44.532,Z 311.847,A -85,B 0,C 180,E1 -29674.583,E2 -29674.583} C_VEL
LIN {X 0,Y 43.973,Z 309.815,A -85,B 0,C 180,E1 -29676.128,E2 -29676.128} C_VEL
LIN {X 0,Y 44.231,Z 309.788,A -85,B 0,C 180,E1 -29682.436,E2 -29682.436} C_VEL
LIN {X 0,Y 44.53,Z 309.751,A -85,B 0,C 180,E1 -29690.912,E2 -29690.912} C_VEL
LIN {X 0,Y 45.141,Z 309.675,A -85,B 0,C 180,E1 -29699.992,E2 -29699.992} C_VEL
LIN {X 0,Y 44.542,Z 309.748,A -85,B 0,C 180,E1 -29709.07,E2 -29709.07} C_VEL
LIN {X 0,Y 44.156,Z 309.792,A -85,B 0,C 180,E1 -29718.553,E2 -29718.553} C_VEL
LIN {X 0,Y 43.848,Z 309.826,A -85,B 0,C 180,E1 -29728.732,E2 -29728.732} C_VEL
LIN {X 0,Y 43.855,Z 309.829,A -85,B 0,C 180,E1 -29739.858,E2 -29739.858} C_VEL
LIN {X 0,Y 43.884,Z 309.823,A -85,B 0,C 180,E1 -29753.187,E2 -29753.187} C_VEL
LIN {X 0,Y 43.851,Z 309.829,A -85,B 0,C 180,E1 -29761.26,E2 -29761.26} C_VEL
LIN {X 0,Y 44.436,Z 309.826,A -85,B 0,C 180,E1 -29774.954,E2 -29774.954} C_VEL
LIN {X 0,Y 45.493,Z 312.636,A -85,B 0,C 180,E1 -29776.942,E2 -29776.942} C_VEL
LIN {X 0,Y 47.28,Z 314.854,A -85,B 0,C 180,E1 -29779.34,E2 -29779.34} C_VEL
LIN {X 0,Y 50.698,Z 320.541,A -85,B 0,C 180,E1 -29783.772,E2 -29783.772} C_VEL
LIN {X 0,Y 54.226,Z 330.507,A -85,B 0,C 180,E1 -29788.407,E2 -29788.407} C_VEL
LIN {X 0,Y 57.267,Z 340.896,A -85,B 0,C 180,E1 -29792.138,E2 -29792.138} C_VEL
LIN {X 0,Y 55.55,Z 357.738,A -85,B 0,C 180,E1 -29794.455,E2 -29794.455} C_VEL
LIN {X 0,Y 54.234,Z 363.482,A -85,B 0,C 180,E1 -29794.933,E2 -29794.933} C_VEL
LIN {X 0,Y 50.329,Z 372.603,A -85,B 0,C 180,E1 -29795.324,E2 -29795.324} C_VEL
LIN {X 0,Y 46.147,Z 381.547,A -85,B 0,C 180,E1 -29796.642,E2 -29796.642} C_VEL
LIN {X 0,Y 44.382,Z 387.018,A -85,B 0,C 180,E1 -29798.627,E2 -29798.627} C_VEL
LIN {X 0,Y 41.808,Z 396.766,A -85,B 0,C 180,E1 -29803.777,E2 -29803.777} C_VEL
LIN {X 0,Y 38.643,Z 407.765,A -85,B 0,C 180,E1 -29812.621,E2 -29812.621} C_VEL
LIN {X 0,Y 36.569,Z 415.899,A -85,B 0,C 180,E1 -29822.049,E2 -29822.049} C_VEL
LIN {X 0,Y 35.207,Z 423.407,A -85,B 0,C 180,E1 -29833.661,E2 -29833.661} C_VEL
LIN {X 0,Y 35.262,Z 430.191,A -85,B 0,C 180,E1 -29846.919,E2 -29846.919} C_VEL
LIN {X 0,Y 37.878,Z 437.298,A -85,B 0,C 180,E1 -29862.984,E2 -29862.984} C_VEL
LIN {X 0,Y 42.33,Z 442.268,A -85,B 0,C 180,E1 -29874.952,E2 -29874.952} C_VEL
LIN {X 0,Y 49.422,Z 446.68,A -85,B 0,C 180,E1 -29885.515,E2 -29885.515} C_VEL
LIN {X 0,Y 57.749,Z 449.885,A -85,B 0,C 180,E1 -29893.207,E2 -29893.207} C_VEL
LIN {X 0,Y 66.767,Z 451.953,A -85,B 0,C 180,E1 -29898.682,E2 -29898.682} C_VEL
LIN {X 0,Y 74.598,Z 452.845,A -85,B 0,C 180,E1 -29902.143,E2 -29902.143} C_VEL
LIN {X 0,Y 69.719,Z 452.814,A -85,B 0,C 180,E1 -29904.879,E2 -29904.879} C_VEL
LIN {X 0,Y 57.878,Z 451.194,A -85,B 0,C 180,E1 -29911.793,E2 -29911.793} C_VEL
LIN {X 0,Y 52.425,Z 449.851,A -85,B 0,C 180,E1 -29916.458,E2 -29916.458} C_VEL
LIN {X 0,Y 45.352,Z 446.913,A -85,B 0,C 180,E1 -29925.79,E2 -29925.79} C_VEL
LIN {X 0,Y 40.196,Z 442.92,A -85,B 0,C 180,E1 -29938.367,E2 -29938.367} C_VEL
LIN {X 0,Y 37.673,Z 437.768,A -85,B 0,C 180,E1 -29953.753,E2 -29953.753} C_VEL
LIN {X 0,Y 37.279,Z 434.66,A -85,B 0,C 180,E1 -29961.874,E2 -29961.874} C_VEL
LIN {X 0,Y 36.589,Z 429.197,A -85,B 0,C 180,E1 -29972.755,E2 -29972.755} C_VEL
LIN {X 0,Y 37.106,Z 421.894,A -85,B 0,C 180,E1 -29984.528,E2 -29984.528} C_VEL
LIN {X 0,Y 38.723,Z 413.935,A -85,B 0,C 180,E1 -29994.393,E2 -29994.393} C_VEL
LIN {X 0,Y 40.669,Z 406.594,A -85,B 0,C 180,E1 -30001.229,E2 -30001.229} C_VEL
LIN {X 0,Y 42.696,Z 398.857,A -85,B 0,C 180,E1 -30006.636,E2 -30006.636} C_VEL
LIN {X 0,Y 45.174,Z 389.223,A -85,B 0,C 180,E1 -30011.393,E2 -30011.393} C_VEL
LIN {X 0,Y 47.395,Z 377.959,A -85,B 0,C 180,E1 -30015.155,E2 -30015.155} C_VEL
LIN {X 0,Y 49.105,Z 362.477,A -85,B 0,C 180,E1 -30018.133,E2 -30018.133} C_VEL
LIN {X 0,Y 48.899,Z 335.504,A -85,B 0,C 180,E1 -30024.321,E2 -30024.321} C_VEL
LIN {X 0,Y 45.313,Z 326.252,A -85,B 0,C 180,E1 -30029.722,E2 -30029.722} C_VEL
LIN {X 0,Y 42.056,Z 319.414,A -85,B 0,C 180,E1 -30035.297,E2 -30035.297} C_VEL
LIN {X 0,Y 39.907,Z 315.908,A -85,B 0,C 180,E1 -30039.368,E2 -30039.368} C_VEL
LIN {X 0,Y 37.553,Z 312.161,A -85,B 0,C 180,E1 -30044.791,E2 -30044.791} C_VEL
LIN {X 0,Y 37.211,Z 310.653,A -85,B 0,C 180,E1 -30046.278,E2 -30046.278} C_VEL
LIN {X 0,Y 37.999,Z 310.564,A -85,B 0,C 180,E1 -30059.991,E2 -30059.991} C_VEL
LIN {X 0,Y 37.336,Z 310.638,A -85,B 0,C 180,E1 -30070.841,E2 -30070.841} C_VEL
LIN {X 0,Y 37.057,Z 310.675,A -85,B 0,C 180,E1 -30078.506,E2 -30078.506} C_VEL
LIN {X 0,Y 36.746,Z 310.716,A -85,B 0,C 180,E1 -30095.002,E2 -30095.002} C_VEL
LIN {X 0,Y 36.768,Z 310.711,A -85,B 0,C 180,E1 -30100.127,E2 -30100.127} C_VEL
LIN {X 0,Y 36.772,Z 310.716,A -85,B 0,C 180,E1 -30109.848,E2 -30109.848} C_VEL
LIN {X 0,Y 36.785,Z 310.706,A -85,B 0,C 180,E1 -30122.747,E2 -30122.747} C_VEL
LIN {X 0,Y 37.781,Z 313.538,A -85,B 0,C 180,E1 -30126.325,E2 -30126.325} C_VEL
LIN {X 0,Y 40.114,Z 315.664,A -85,B 0,C 180,E1 -30131.035,E2 -30131.035} C_VEL
LIN {X 0,Y 43.387,Z 320.799,A -85,B 0,C 180,E1 -30136.912,E2 -30136.912} C_VEL
LIN {X 0,Y 45.656,Z 324.824,A -85,B 0,C 180,E1 -30140.368,E2 -30140.368} C_VEL
LIN {X 0,Y 48.597,Z 333.663,A -85,B 0,C 180,E1 -30145.145,E2 -30145.145} C_VEL
LIN {X 0,Y 50.802,Z 341.484,A -85,B 0,C 180,E1 -30148.51,E2 -30148.51} C_VEL
LIN {X 0,Y 49.197,Z 357.634,A -85,B 0,C 180,E1 -30151.015,E2 -30151.015} C_VEL
LIN {X 0,Y 47.195,Z 373.217,A -85,B 0,C 180,E1 -30153.844,E2 -30153.844} C_VEL
LIN {X 0,Y 45.031,Z 384.203,A -85,B 0,C 180,E1 -30157.449,E2 -30157.449} C_VEL
LIN {X 0,Y 44.382,Z 387.018,A -85,B 0,C 180,E1 -30158.627,E2 -30158.627} C_VEL
LIN {X 0,Y 42.451,Z 392.318,A -85,B 0,C 180,E1 -30160.877,E2 -30160.877} C_VEL
LIN {X 0,Y 37.452,Z 400.348,A -85,B 0,C 180,E1 -30165.057,E2 -30165.057} C_VEL
LIN {X 0,Y 33.182,Z 406.523,A -85,B 0,C 180,E1 -30169.967,E2 -30169.967} C_VEL
LIN {X 0,Y 30.712,Z 411.03,A -85,B 0,C 180,E1 -30175.243,E2 -30175.243} C_VEL
LIN {X 0,Y 30.162,Z 412.569,A -85,B 0,C 180,E1 -30177.322,E2 -30177.322} C_VEL
LIN {X 0,Y 28.368,Z 421.066,A -85,B 0,C 180,E1 -30192.012,E2 -30192.012} C_VEL
LIN {X 0,Y 28.55,Z 429.076,A -85,B 0,C 180,E1 -30210.52,E2 -30210.52} C_VEL
LIN {X 0,Y 31.373,Z 435.486,A -85,B 0,C 180,E1 -30227.066,E2 -30227.066} C_VEL
LIN {X 0,Y 36.17,Z 440.612,A -85,B 0,C 180,E1 -30240.009,E2 -30240.009} C_VEL
LIN {X 0,Y 42.805,Z 444.99,A -85,B 0,C 180,E1 -30249.915,E2 -30249.915} C_VEL
LIN {X 0,Y 51.688,Z 448.896,A -85,B 0,C 180,E1 -30257.874,E2 -30257.874} C_VEL
LIN {X 0,Y 58.869,Z 450.965,A -85,B 0,C 180,E1 -30262.088,E2 -30262.088} C_VEL
LIN {X 0,Y 57.434,Z 450.736,A -85,B 0,C 180,E1 -30263.808,E2 -30263.808} C_VEL
LIN {X 0,Y 48.609,Z 448.514,A -85,B 0,C 180,E1 -30269.838,E2 -30269.838} C_VEL
LIN {X 0,Y 40.671,Z 445.313,A -85,B 0,C 180,E1 -30278.963,E2 -30278.963} C_VEL
LIN {X 0,Y 34.539,Z 441.08,A -85,B 0,C 180,E1 -30292.384,E2 -30292.384} C_VEL
LIN {X 0,Y 31.245,Z 435.638,A -85,B 0,C 180,E1 -30310.285,E2 -30310.285} C_VEL
LIN {X 0,Y 30.87,Z 433.436,A -85,B 0,C 180,E1 -30316.844,E2 -30316.844} C_VEL
LIN {X 0,Y 29.815,Z 427.906,A -85,B 0,C 180,E1 -30330.003,E2 -30330.003} C_VEL
LIN {X 0,Y 30.077,Z 421.079,A -85,B 0,C 180,E1 -30343.516,E2 -30343.516} C_VEL
LIN {X 0,Y 31.592,Z 413.591,A -85,B 0,C 180,E1 -30354.999,E2 -30354.999} C_VEL
LIN {X 0,Y 33.821,Z 405.769,A -85,B 0,C 180,E1 -30363.76,E2 -30363.76} C_VEL
LIN {X 0,Y 36.36,Z 396.896,A -85,B 0,C 180,E1 -30370.722,E2 -30370.722} C_VEL
LIN {X 0,Y 39.369,Z 385.844,A -85,B 0,C 180,E1 -30376.405,E2 -30376.405} C_VEL
LIN {X 0,Y 41.42,Z 374.918,A -85,B 0,C 180,E1 -30379.856,E2 -30379.856} C_VEL
LIN {X 0,Y 42.883,Z 361.744,A -85,B 0,C 180,E1 -30382.565,E2 -30382.565} C_VEL
LIN {X 0,Y 43.031,Z 337.5,A -85,B 0,C 180,E1 -30388.961,E2 -30388.961} C_VEL
LIN {X 0,Y 39.817,Z 328.777,A -85,B 0,C 180,E1 -30395.206,E2 -30395.206} C_VEL
LIN {X 0,Y 37.359,Z 323.69,A -85,B 0,C 180,E1 -30400.612,E2 -30400.612} C_VEL
LIN {X 0,Y 35.209,Z 319.773,A -85,B 0,C 180,E1 -30406.341,E2 -30406.341} C_VEL
LIN {X 0,Y 33.647,Z 316.675,A -85,B 0,C 180,E1 -30411.733,E2 -30411.733} C_VEL
LIN {X 0,Y 31.938,Z 314.678,A -85,B 0,C 180,E1 -30418.413,E2 -30418.413} C_VEL
LIN {X 0,Y 31.327,Z 313.64,A -85,B 0,C 180,E1 -30421.596,E2 -30421.596} C_VEL
LIN {X 0,Y 30.338,Z 311.601,A -85,B 0,C 180,E1 -30428.733,E2 -30428.733} C_VEL
LIN {X 0,Y 29.866,Z 311.45,A -85,B 0,C 180,E1 -30439.725,E2 -30439.725} C_VEL
LIN {X 0,Y 29.691,Z 311.654,A -85,B 0,C 180,E1 -30456.005,E2 -30456.005} C_VEL
LIN {X 0,Y 30.89,Z 314.834,A -85,B 0,C 180,E1 -30467.656,E2 -30467.656} C_VEL
LIN {X 0,Y 33.665,Z 317.375,A -85,B 0,C 180,E1 -30478.835,E2 -30478.835} C_VEL
LIN {X 0,Y 35.419,Z 320.404,A -85,B 0,C 180,E1 -30484.476,E2 -30484.476} C_VEL
LIN {X 0,Y 37.027,Z 322.232,A -85,B 0,C 180,E1 -30488.386,E2 -30488.386} C_VEL
LIN {X 0,Y 40.434,Z 328.07,A -85,B 0,C 180,E1 -30495.561,E2 -30495.561} C_VEL
LIN {X 0,Y 43.037,Z 336.502,A -85,B 0,C 180,E1 -30500.957,E2 -30500.957} C_VEL
LIN {X 0,Y 44.722,Z 342.966,A -85,B 0,C 180,E1 -30504.211,E2 -30504.211} C_VEL
LIN {X 0,Y 41.397,Z 370.094,A -85,B 0,C 180,E1 -30508.943,E2 -30508.943} C_VEL
LIN {X 0,Y 39.04,Z 382.057,A -85,B 0,C 180,E1 -30512.577,E2 -30512.577} C_VEL
LIN {X 0,Y 36.256,Z 392.656,A -85,B 0,C 180,E1 -30518.021,E2 -30518.021} C_VEL
LIN {X 0,Y 33.447,Z 401.428,A -85,B 0,C 180,E1 -30524.572,E2 -30524.572} C_VEL
LIN {X 0,Y 31.299,Z 408.612,A -85,B 0,C 180,E1 -30532.172,E2 -30532.172} C_VEL
LIN {X 0,Y 30.162,Z 412.569,A -85,B 0,C 180,E1 -30537.322,E2 -30537.322} C_VEL
LIN {X 0,Y 28.288,Z 416.961,A -85,B 0,C 180,E1 -30544.154,E2 -30544.154} C_VEL
LIN {X 0,Y 25.938,Z 420.846,A -85,B 0,C 180,E1 -30552.311,E2 -30552.311} C_VEL
LIN {X 0,Y 22.886,Z 428.895,A -85,B 0,C 180,E1 -30578.51,E2 -30578.51} C_VEL
LIN {X 0,Y 24.257,Z 432.358,A -85,B 0,C 180,E1 -30589.853,E2 -30589.853} C_VEL
LIN {X 0,Y 30.713,Z 439.046,A -85,B 0,C 180,E1 -30607.574,E2 -30607.574} C_VEL
LIN {X 0,Y 38.747,Z 444.109,A -85,B 0,C 180,E1 -30617.989,E2 -30617.989} C_VEL
LIN {X 0,Y 43.355,Z 446.377,A -85,B 0,C 180,E1 -30621.804,E2 -30621.804} C_VEL
LIN {X 0,Y 39.546,Z 444.914,A -85,B 0,C 180,E1 -30627.312,E2 -30627.312} C_VEL
LIN {X 0,Y 31.641,Z 440.729,A -85,B 0,C 180,E1 -30638.981,E2 -30638.981} C_VEL
LIN {X 0,Y 26.045,Z 435.417,A -85,B 0,C 180,E1 -30657.343,E2 -30657.343} C_VEL
LIN {X 0,Y 24.313,Z 430.939,A -85,B 0,C 180,E1 -30673.203,E2 -30673.203} C_VEL
LIN {X 0,Y 22.963,Z 424.968,A -85,B 0,C 180,E1 -30690.004,E2 -30690.004} C_VEL
LIN {X 0,Y 23.789,Z 415.795,A -85,B 0,C 180,E1 -30711.219,E2 -30711.219} C_VEL
LIN {X 0,Y 26.471,Z 406.654,A -85,B 0,C 180,E1 -30725.216,E2 -30725.216} C_VEL
LIN {X 0,Y 29.263,Z 397.979,A -85,B 0,C 180,E1 -30733.888,E2 -30733.888} C_VEL
LIN {X 0,Y 32.158,Z 388.595,A -85,B 0,C 180,E1 -30739.901,E2 -30739.901} C_VEL
LIN {X 0,Y 34.824,Z 377.551,A -85,B 0,C 180,E1 -30744.417,E2 -30744.417} C_VEL
LIN {X 0,Y 36.861,Z 363.14,A -85,B 0,C 180,E1 -30747.763,E2 -30747.763} C_VEL
LIN {X 0,Y 37.491,Z 339.763,A -85,B 0,C 180,E1 -30754.673,E2 -30754.673} C_VEL
LIN {X 0,Y 34.605,Z 331.082,A -85,B 0,C 180,E1 -30762.635,E2 -30762.635} C_VEL
LIN {X 0,Y 31.895,Z 325.103,A -85,B 0,C 180,E1 -30772.074,E2 -30772.074} C_VEL
LIN {X 0,Y 30.714,Z 322.57,A -85,B 0,C 180,E1 -30777.53,E2 -30777.53} C_VEL
LIN {X 0,Y 28.65,Z 318.342,A -85,B 0,C 180,E1 -30793.01,E2 -30793.01} C_VEL
LIN {X 0,Y 28.271,Z 318.614,A -85,B 0,C 180,E1 -30812.609,E2 -30812.609} C_VEL
LIN {X 0,Y 29.099,Z 321.479,A -85,B 0,C 180,E1 -30824.424,E2 -30824.424} C_VEL
LIN {X 0,Y 30.879,Z 323.582,A -85,B 0,C 180,E1 -30834.029,E2 -30834.029} C_VEL
LIN {X 0,Y 33.014,Z 327.013,A -85,B 0,C 180,E1 -30842.066,E2 -30842.066} C_VEL
LIN {X 0,Y 35.327,Z 331.222,A -85,B 0,C 180,E1 -30848.895,E2 -30848.895} C_VEL
LIN {X 0,Y 36.12,Z 333.158,A -85,B 0,C 180,E1 -30851.048,E2 -30851.048} C_VEL
LIN {X 0,Y 38.119,Z 341.147,A -85,B 0,C 180,E1 -30856.815,E2 -30856.815} C_VEL
LIN {X 0,Y 38.852,Z 344.51,A -85,B 0,C 180,E1 -30858.807,E2 -30858.807} C_VEL
LIN {X 0,Y 35.212,Z 370.851,A -85,B 0,C 180,E1 -30863.59,E2 -30863.59} C_VEL
LIN {X 0,Y 32.287,Z 383.731,A -85,B 0,C 180,E1 -30868.006,E2 -30868.006} C_VEL
LIN {X 0,Y 29.349,Z 393.541,A -85,B 0,C 180,E1 -30873.82,E2 -30873.82} C_VEL
LIN {X 0,Y 26.275,Z 402.215,A -85,B 0,C 180,E1 -30881.622,E2 -30881.622} C_VEL
LIN {X 0,Y 23.634,Z 410.253,A -85,B 0,C 180,E1 -30892.728,E2 -30892.728} C_VEL
LIN {X 0,Y 21.67,Z 418.044,A -85,B 0,C 180,E1 -30908.512,E2 -30908.512} C_VEL
LIN {X 0,Y 21.572,Z 426.059,A -85,B 0,C 180,E1 -30930.706,E2 -30930.706} C_VEL
LIN {X 0,Y 24.257,Z 432.358,A -85,B 0,C 180,E1 -30949.853,E2 -30949.853} C_VEL
LIN {X 0,Y 24.617,Z 433.607,A -85,B 0,C 180,E1 -30954.754,E2 -30954.754} C_VEL
LIN {X 0,Y 23.981,Z 434.547,A -85,B 0,C 180,E1 -30962.415,E2 -30962.415} C_VEL
LIN {X 0,Y 22.436,Z 434.781,A -85,B 0,C 180,E1 -30973.481,E2 -30973.481} C_VEL
LIN {X 0,Y 20.482,Z 433.938,A -85,B 0,C 180,E1 -30988.742,E2 -30988.742} C_VEL
LIN {X 0,Y 19.115,Z 432.063,A -85,B 0,C 180,E1 -31006.793,E2 -31006.793} C_VEL
LIN {X 0,Y 18.507,Z 430.207,A -85,B 0,C 180,E1 -31018.415,E2 -31018.415} C_VEL
LIN {X 0,Y 17.649,Z 427.728,A -85,B 0,C 180,E1 -31028.945,E2 -31028.945} C_VEL
LIN {X 0,Y 16.076,Z 420.019,A -85,B 0,C 180,E1 -31056.281,E2 -31056.281} C_VEL
LIN {X 0,Y 17.316,Z 412.726,A -85,B 0,C 180,E1 -31077.174,E2 -31077.174} C_VEL
LIN {X 0,Y 19.957,Z 405.231,A -85,B 0,C 180,E1 -31091.327,E2 -31091.327} C_VEL
LIN {X 0,Y 23.39,Z 395.907,A -85,B 0,C 180,E1 -31101.93,E2 -31101.93} C_VEL
LIN {X 0,Y 27.286,Z 384.33,A -85,B 0,C 180,E1 -31109.077,E2 -31109.077} C_VEL
LIN {X 0,Y 29.604,Z 374.184,A -85,B 0,C 180,E1 -31112.692,E2 -31112.692} C_VEL
LIN {X 0,Y 31.322,Z 362.074,A -85,B 0,C 180,E1 -31115.576,E2 -31115.576} C_VEL
LIN {X 0,Y 32.403,Z 342.065,A -85,B 0,C 180,E1 -31122.231,E2 -31122.231} C_VEL
LIN {X 0,Y 30.518,Z 334.936,A -85,B 0,C 180,E1 -31130.461,E2 -31130.461} C_VEL
LIN {X 0,Y 28.454,Z 328.971,A -85,B 0,C 180,E1 -31142.117,E2 -31142.117} C_VEL
LIN {X 0,Y 27.213,Z 325.484,A -85,B 0,C 180,E1 -31155.658,E2 -31155.658} C_VEL
LIN {X 0,Y 26.944,Z 325.648,A -85,B 0,C 180,E1 -31168.975,E2 -31168.975} C_VEL
LIN {X 0,Y 28.48,Z 329.979,A -85,B 0,C 180,E1 -31189.108,E2 -31189.108} C_VEL
LIN {X 0,Y 30.698,Z 334.186,A -85,B 0,C 180,E1 -31199.848,E2 -31199.848} C_VEL
LIN {X 0,Y 31.859,Z 337.347,A -85,B 0,C 180,E1 -31204.395,E2 -31204.395} C_VEL
LIN {X 0,Y 33.432,Z 345.824,A -85,B 0,C 180,E1 -31211.453,E2 -31211.453} C_VEL
LIN {X 0,Y 29.677,Z 370.395,A -85,B 0,C 180,E1 -31215.768,E2 -31215.768} C_VEL
LIN {X 0,Y 27.013,Z 381.576,A -85,B 0,C 180,E1 -31219.216,E2 -31219.216} C_VEL
LIN {X 0,Y 23.336,Z 392.79,A -85,B 0,C 180,E1 -31225.788,E2 -31225.788} C_VEL
LIN {X 0,Y 19.424,Z 402.472,A -85,B 0,C 180,E1 -31235.921,E2 -31235.921} C_VEL
LIN {X 0,Y 16.682,Z 409.56,A -85,B 0,C 180,E1 -31248.639,E2 -31248.639} C_VEL
LIN {X 0,Y 14.697,Z 416.863,A -85,B 0,C 180,E1 -31269.416,E2 -31269.416} C_VEL
LIN {X 0,Y 14.681,Z 422.632,A -85,B 0,C 180,E1 -31291.426,E2 -31291.426} C_VEL
LIN {X 0,Y 17.411,Z 428.88,A -85,B 0,C 180,E1 -31315.435,E2 -31315.435} C_VEL
LIN {X 0,Y 23.121,Z 434.95,A -85,B 0,C 180,E1 -31332.969,E2 -31332.969} C_VEL
LIN {X 0,Y 30.743,Z 440.349,A -85,B 0,C 180,E1 -31343.886,E2 -31343.886} C_VEL
LIN {X 0,Y 21.832,Z 434.243,A -85,B 0,C 180,E1 -31362.74,E2 -31362.74} C_VEL
LIN {X 0,Y 18.624,Z 429.645,A -85,B 0,C 180,E1 -31381.861,E2 -31381.861} C_VEL
LIN {X 0,Y 17.649,Z 427.728,A -85,B 0,C 180,E1 -31388.945,E2 -31388.945} C_VEL
LIN {X 0,Y 15.856,Z 423.816,A -85,B 0,C 180,E1 -31401.946,E2 -31401.946} C_VEL
LIN {X 0,Y 14.061,Z 419.506,A -85,B 0,C 180,E1 -31415.567,E2 -31415.567} C_VEL
LIN {X 0,Y 12.628,Z 408.253,A -85,B 0,C 180,E1 -31452.368,E2 -31452.368} C_VEL
LIN {X 0,Y 14.228,Z 403.015,A -85,B 0,C 180,E1 -31464.121,E2 -31464.121} C_VEL
LIN {X 0,Y 19.192,Z 391.474,A -85,B 0,C 180,E1 -31476.446,E2 -31476.446} C_VEL
LIN {X 0,Y 22.578,Z 381.842,A -85,B 0,C 180,E1 -31480.903,E2 -31480.903} C_VEL
LIN {X 0,Y 24.945,Z 372.117,A -85,B 0,C 180,E1 -31483.763,E2 -31483.763} C_VEL
LIN {X 0,Y 26.54,Z 361.835,A -85,B 0,C 180,E1 -31486.121,E2 -31486.121} C_VEL
LIN {X 0,Y 27.99,Z 343.877,A -85,B 0,C 180,E1 -31492.853,E2 -31492.853} C_VEL
LIN {X 0,Y 27.047,Z 338.832,A -85,B 0,C 180,E1 -31500.307,E2 -31500.307} C_VEL
LIN {X 0,Y 26.163,Z 334.512,A -85,B 0,C 180,E1 -31510.536,E2 -31510.536} C_VEL
LIN {X 0,Y 25.856,Z 332.391,A -85,B 0,C 180,E1 -31519.11,E2 -31519.11} C_VEL
LIN {X 0,Y 25.674,Z 332.895,A -85,B 0,C 180,E1 -31526.504,E2 -31526.504} C_VEL
LIN {X 0,Y 26.332,Z 336.206,A -85,B 0,C 180,E1 -31543.157,E2 -31543.157} C_VEL
LIN {X 0,Y 27.695,Z 339.851,A -85,B 0,C 180,E1 -31553.565,E2 -31553.565} C_VEL
LIN {X 0,Y 28.381,Z 344.314,A -85,B 0,C 180,E1 -31558.995,E2 -31558.995} C_VEL
LIN {X 0,Y 28.662,Z 346.946,A -85,B 0,C 180,E1 -31561.402,E2 -31561.402} C_VEL
LIN {X 0,Y 24.735,Z 370.351,A -85,B 0,C 180,E1 -31564.872,E2 -31564.872} C_VEL
LIN {X 0,Y 21.823,Z 381.469,A -85,B 0,C 180,E1 -31567.705,E2 -31567.705} C_VEL
LIN {X 0,Y 17.687,Z 392.574,A -85,B 0,C 180,E1 -31573.373,E2 -31573.373} C_VEL
LIN {X 0,Y 13.239,Z 401.997,A -85,B 0,C 180,E1 -31583.439,E2 -31583.439} C_VEL
LIN {X 0,Y 9.534,Z 409.752,A -85,B 0,C 180,E1 -31602.482,E2 -31602.482} C_VEL
LIN {X 0,Y 7.637,Z 416.971,A -85,B 0,C 180,E1 -31640.862,E2 -31640.862} C_VEL
LIN {X 0,Y 9.766,Z 423.269,A -85,B 0,C 180,E1 -31680.035,E2 -31680.035} C_VEL
LIN {X 0,Y 16.84,Z 430.756,A -85,B 0,C 180,E1 -31704.688,E2 -31704.688} C_VEL
LIN {X 0,Y 16.49,Z 430.464,A -85,B 0,C 180,E1 -31711.541,E2 -31711.541} C_VEL
LIN {X 0,Y 13.118,Z 426.831,A -85,B 0,C 180,E1 -31727.969,E2 -31727.969} C_VEL
LIN {X 0,Y 9.616,Z 420.26,A -85,B 0,C 180,E1 -31759.483,E2 -31759.483} C_VEL
LIN {X 0,Y 9.911,Z 413.165,A -85,B 0,C 180,E1 -31796.319,E2 -31796.319} C_VEL
LIN {X 0,Y 12.862,Z 405.93,A -85,B 0,C 180,E1 -31818.717,E2 -31818.717} C_VEL
LIN {X 0,Y 14.228,Z 403.015,A -85,B 0,C 180,E1 -31824.121,E2 -31824.121} C_VEL
LIN {X 0,Y 16.062,Z 397.854,A -85,B 0,C 180,E1 -31832.613,E2 -31832.613} C_VEL
LIN {X 0,Y 17.281,Z 392.523,A -85,B 0,C 180,E1 -31840.706,E2 -31840.706} C_VEL
LIN {X 0,Y 19.206,Z 381.477,A -85,B 0,C 180,E1 -31854.132,E2 -31854.132} C_VEL
LIN {X 0,Y 19.899,Z 377.659,A -85,B 0,C 180,E1 -31856.91,E2 -31856.91} C_VEL
LIN {X 0,Y 20.654,Z 373.775,A -85,B 0,C 180,E1 -31858.372,E2 -31858.372} C_VEL
LIN {X 0,Y 22.731,Z 362.647,A -85,B 0,C 180,E1 -31859.985,E2 -31859.985} C_VEL
LIN {X 0,Y 24.69,Z 346.099,A -85,B 0,C 180,E1 -31866.291,E2 -31866.291} C_VEL
LIN {X 0,Y 24.547,Z 342.929,A -85,B 0,C 180,E1 -31872.208,E2 -31872.208} C_VEL
LIN {X 0,Y 24.527,Z 340.104,A -85,B 0,C 180,E1 -31880.189,E2 -31880.189} C_VEL
LIN {X 0,Y 24.513,Z 339.845,A -85,B 0,C 180,E1 -31882.707,E2 -31882.707} C_VEL
LIN {X 0,Y 24.498,Z 342.239,A -85,B 0,C 180,E1 -31895.626,E2 -31895.626} C_VEL
LIN {X 0,Y 24.96,Z 345.022,A -85,B 0,C 180,E1 -31904.38,E2 -31904.38} C_VEL
LIN {X 0,Y 25.003,Z 348.471,A -85,B 0,C 180,E1 -31908.444,E2 -31908.444} C_VEL
LIN {X 0,Y 20.88,Z 371.025,A -85,B 0,C 180,E1 -31909.605,E2 -31909.605} C_VEL
LIN {X 0,Y 17.454,Z 382.987,A -85,B 0,C 180,E1 -31910.502,E2 -31910.502} C_VEL
LIN {X 0,Y 12.901,Z 393.612,A -85,B 0,C 180,E1 -31911.889,E2 -31911.889} C_VEL
LIN {X 0,Y 7.535,Z 403.243,A -85,B 0,C 180,E1 -31915.412,E2 -31915.412} C_VEL
LIN {X 0,Y 2.214,Z 411.032,A -85,B 0,C 180,E1 -31932.676,E2 -31932.676} C_VEL
LIN {X 0,Y 2.47,Z 416.328,A -85,B 0,C 180,E1 -32069.985,E2 -32069.985} C_VEL
LIN {X 0,Y 2.463,Z 414.669,A -85,B 0,C 180,E1 -32130.04,E2 -32130.04} C_VEL
LIN {X 0,Y 7.293,Z 405.107,A -85,B 0,C 180,E1 -32204.561,E2 -32204.561} C_VEL
LIN {X 0,Y 12.383,Z 395.998,A -85,B 0,C 180,E1 -32213.377,E2 -32213.377} C_VEL
LIN {X 0,Y 16.79,Z 386.203,A -85,B 0,C 180,E1 -32216.328,E2 -32216.328} C_VEL
LIN {X 0,Y 20.481,Z 374.633,A -85,B 0,C 180,E1 -32218.214,E2 -32218.214} C_VEL
LIN {X 0,Y 20.654,Z 373.775,A -85,B 0,C 180,E1 -32218.372,E2 -32218.372} C_VEL
LIN {X 0,Y 21.146,Z 369.947,A -85,B 0,C 180,E1 -32220.769,E2 -32220.769} C_VEL
LIN {X 0,Y 21.208,Z 363.996,A -85,B 0,C 180,E1 -32229.189,E2 -32229.189} C_VEL
LIN {X 0,Y 21.6,Z 358.044,A -85,B 0,C 180,E1 -32237.954,E2 -32237.954} C_VEL
LIN {X 0,Y 22.149,Z 354.188,A -85,B 0,C 180,E1 -32240.567,E2 -32240.567} C_VEL
LIN {X 0,Y 23.06,Z 348.54,A -85,B 0,C 180,E1 -32242.364,E2 -32242.364} C_VEL
LIN {X 0,Y 23.177,Z 347.745,A -85,B 0,C 180,E1 -32244.528,E2 -32244.528} C_VEL
LIN {X 0,Y 23.052,Z 349.467,A -85,B 0,C 180,E1 -32251.586,E2 -32251.586} C_VEL
LIN {X 0,Y 19.686,Z 368.673,A -85,B 0,C 180,E1 -32250.213,E2 -32250.213} C_VEL
LIN {X 0,Y 17.131,Z 378.896,A -85,B 0,C 180,E1 -32247.828,E2 -32247.828} C_VEL
LIN {X 0,Y 15.646,Z 383.725,A -85,B 0,C 180,E1 -32246.042,E2 -32246.042} C_VEL
LIN {X 0,Y 15.065,Z 385.36,A -85,B 0,C 180,E1 -32241.076,E2 -32241.076} C_VEL
LIN {X 0,Y 18.764,Z 373.157,A -85,B 0,C 180,E1 -32238.301,E2 -32238.301} C_VEL
LIN {X 0,Y 20.794,Z 362.767,A -85,B 0,C 180,E1 -32237.999,E2 -32237.999} C_VEL
LIN {X 0,Y 22.149,Z 354.188,A -85,B 0,C 180,E1 -32240.567,E2 -32240.567} C_VEL
LIN {X 0,Y 25.7,Z 354.551,A -85,B 0,C 180,E1 -32244.817,E2 -32244.817} C_VEL
LIN {X 0,Y 25.7,Z 600,A -85,B 0,C 180,E1 -32244.817,E2 -32244.817} C_VEL
LIN {X 0,Y 25.7,Z 600,A -85,B 0,C 180,E1 -32244.817,E2 -32244.817}

QRS_NEXT_CUT()

QRS_NEXT()
QRS_HOME()

END
